	THIS^.assertorContainer.assertor.assert.strings.unicode.lengthIsExact(
		stringToCheck := stringToTest,
		expectedLength := expectedLength,
		stringLengthUnit := CNM_AssertionInterfaces.UnicodeStringLengthUnit.CHARACTERS_NFC,
		message			:= ''
	);
	
	THIS^.AssertEquals_BOOL(
		Expected 	:= assertionIsWrong,
		Actual 		:= THIS^.assertorContainer.wasAssertionWrong,
		Message 	:= messageStringBuilder.sOut
	);

	THIS^.AssertEquals_WSTRING(
		Expected 	:= stringToTestBeforeAssertion,
		Actual 		:= stringToTest,
		Message 	:= 'the assertion changed $'stringToTest$''
	);
	
CNM_AssertionInterfaces.UnicodeStringLengthUnit.VISIBLE_CHARACTERS:	
	currentStringLengthUnit := 'VISIBLE_CHARACTERS';
	
	assertionIsWrong := stringToTestVisibleCharacters <> expectedLength;
	
	message := SEL(
		assertionIsWrong,
		'stringToCheck is $'%s$' with expectedLength %u assertion must be TRUE  (%S)', 
		'stringToCheck is $'%s$' with expectedLength %u assertion must be FALSE  (%S)'
	);
	
	messageStringBuilder(
		sFormat := message,
		arg1 := THIS^.AnyToArg(stringToTestAsString),
		arg2 := THIS^.AnyToArg(expectedLength),
		arg3 := THIS^.AnyToArg(currentStringLengthUnit)
	);
	
	THIS^.assertorContainer.assertor.assert.strings.unicode.lengthIsExact(
		stringToCheck := stringToTest,
		expectedLength := expectedLength,
		stringLengthUnit := CNM_AssertionInterfaces.UnicodeStringLengthUnit.VISIBLE_CHARACTERS,
		message			:= ''
	);
	
	THIS^.AssertEquals_BOOL(
		Expected 	:= assertionIsWrong,
		Actual 		:= THIS^.assertorContainer.wasAssertionWrong,
		Message 	:= messageStringBuilder.sOut
	);

	THIS^.AssertEquals_WSTRING(
		Expected 	:= stringToTestBeforeAssertion,
		Actual 		:= stringToTest,
		Message 	:= 'the assertion changed $'stringToTest$''
	);
	
CNM_AssertionInterfaces.UnicodeStringLengthUnit.WIDTH:	
	currentStringLengthUnit := 'WIDTH';
	
	assertionIsWrong := TO_UDINT(stringToTestWidth) <> expectedLength;
	
	message := SEL(
		assertionIsWrong,
		'stringToCheck is $'%s$' with expectedLength %u assertion must be TRUE  (%S)', 
		'stringToCheck is $'%s$' with expectedLength %u assertion must be FALSE  (%S)'
	);
	
	messageStringBuilder(
		sFormat := message,
		arg1 := THIS^.AnyToArg(stringToTestAsString),
		arg2 := THIS^.AnyToArg(expectedLength),
		arg3 := THIS^.AnyToArg(currentStringLengthUnit)
	);
	
	THIS^.assertorContainer.assertor.assert.strings.unicode.lengthIsExact(
		stringToCheck := stringToTest,
		expectedLength := expectedLength,
		stringLengthUnit := CNM_AssertionInterfaces.UnicodeStringLengthUnit.WIDTH,
		message			:= ''
	);
	
	THIS^.AssertEquals_BOOL(
		Expected 	:= assertionIsWrong,
		Actual 		:= THIS^.assertorContainer.wasAssertionWrong,
		Message 	:= messageStringBuilder.sOut
	);

	THIS^.AssertEquals_WSTRING(
		Expected 	:= stringToTestBeforeAssertion,
		Actual 		:= stringToTest,
		Message 	:= 'the assertion changed $'stringToTest$''
	);

END_CASE
END_METHOD

(*
short summary
==================
This test method tests ``assert.string.unicode.lengthIsMax``
method of CNM_AssertionInterfaces library with various inputs

.. <legal notes>

legal notes
=================
| SPDX-FileCopyrightText: © 2022 ekvip automation GmbH <info@ekvip.de>
| SPDX-License-Identifier: Apache-2.0
| For details check: Apache-2.0_

.. _Apache-2.0: https://www.apache.org/licenses/LICENSE-2.0

.. </legal notes>

*)


METHOD testLengthIsMax : BOOL
VAR_INPUT
	(* for the test it's the parameter ``stringToCheck`` *)
	stringToTest 			:WSTRING(Tc2_System.MAX_STRING_LENGTH);
	(* for the test it's the parameter ``maxLength`` *)
	expectedLength 			:UDINT;
	(* UnicodeStringLengthUnit the input is tested for *)
	stringLengthUnit		:CNM_AssertionInterfaces.UnicodeStringLengthUnit;
	(* contains ``stringToTest`` in only ascii charachters for test output *)
	stringToTestPrintable	:Tc2_System.T_MaxString := '';
END_VAR
VAR 
	(* just the expectation if the assertion to test must be worng or true *)
	assertionIsWrong					:BOOL;
	(* contains the format string for the test message *)
	message								:Tc2_System.T_MaxString;
	(* used for placeholder string if stringToTest can't be printed *)
	stringToTestAsString 				:Tc2_System.T_MaxString;
	(* holds string with current ´´stringLengthUnit´´ for the test message*)
	currentStringLengthUnit 			:Tc2_System.T_MaxString;
	(* TwinCAT printf with the test message *)
	messageStringBuilder				:Tc2_Utilities.FB_FormatString;
	(* length of current string to check in bytes *)
	stringToTestByteCount				:UDINT;
	(* count of words in current string *)
	stringToTestWordCount				:UDINT;
	(* length of current string to check in characters *)
	stringToTestCodePointCount			:UDINT;
	(* length of ´´stringToCheck´´ *)
	normalizedLength 					:UDINT;
	(* holds the normalized ´´stringToCheck´´ *)
	normalizedStringToTest 				:WSTRING(Tc2_System.MAX_STRING_LENGTH);
	(* width of ´´stringToCheck´´ *)
	stringToTestWidth 					:DINT;
	(* visible characters of ´´stringToCheck´´ *)
	stringToTestVisibleCharacters 		:UDINT := 0;
	(*string in UTF32*)
	utf32String							:ARRAY [0..Tc2_System.Global_Variables.MAX_STRING_LENGTH]  OF CNM_UnicodeUtilities.UnicodeCodePoint;
	(* utf32 code point count *)
	utf32CodePointCount 				:UDINT;
	(* bytes in utf8 string *)
	utf8ByteCount 						:UDINT;
	(* hold stringToCheck before assertion *)
	stringToTestBeforeAssertion			:WSTRING(Tc2_System.MAX_STRING_LENGTH);
END_VAR
THIS^.assertorContainer.resetAssertor();

stringToTestBeforeAssertion := stringToTest;

CNM_UnicodeUtilities.GetUtf16StringLength(ADR(stringToTest), wordCount => stringToTestWordCount, characterCount => stringToTestCodePointCount,);
CNM_UnicodeUtilities.GetUtf16StringWidth(ADR(stringToTest), visibleCharacters => stringToTestVisibleCharacters, width => stringToTestWidth);
stringToTestByteCount := stringToTestWordCount * 2;

CNM_UnicodeUtilities.GetCodepointsFromUtf16String(
	utf16StringAddress := ADR(stringToTest),
	utf16StringWordCount := stringToTestWordCount,
	codepointBuffer :=ADR(utf32String),
	bufferSize := SIZEOF(utf32String),
	codePointCount => utf32CodePointCount
);

CNM_UnicodeUtilities.GetUtf8StringFromCodepoints(
	addressOfCodePoints := ADR(utf32String),
	codePointCount := utf32CodePointCount,
	utf8StringBuffer := ADR(stringToTestAsString),
	bufferSize := MAX_STRING_LENGTH + 1,
	utf8StringByteCount => utf8ByteCount
);

IF ( Tc2_Standard.LEN(stringToTestPrintable) <> 0 ) THEN
	stringToTestAsString := stringToTestPrintable;
END_IF


CASE stringLengthUnit OF
	
CNM_AssertionInterfaces.UnicodeStringLengthUnit.BYTES:
	currentStringLengthUnit := 'BYTES';
	
	assertionIsWrong := stringToTestByteCount > expectedLength;
	
	message := SEL(
		assertionIsWrong,
		'stringToCheck is $'%s$' with expectedLength %u assertion must be TRUE  (%S)', 
		'stringToCheck is $'%s$' with expectedLength %u assertion must be FALSE  (%S)'
	);
	
	messageStringBuilder(
		sFormat := message,
		arg1 := THIS^.AnyToArg(stringToTestAsString),
		arg2 := THIS^.AnyToArg(expectedLength),
		arg3 := THIS^.AnyToArg(currentStringLengthUnit)
	);
	
	THIS^.assertorContainer.assertor.assert.strings.unicode.lengthIsMax(
		stringToCheck := stringToTest,
		maxLength := expectedLength,
		stringLengthUnit := CNM_AssertionInterfaces.UnicodeStringLengthUnit.BYTES,
		message			:= ''
	);
	
	THIS^.AssertEquals_BOOL(
		Expected 	:= assertionIsWrong,
		Actual 		:= THIS^.assertorContainer.wasAssertionWrong,
		Message 	:= messageStringBuilder.sOut
	);

	THIS^.AssertEquals_WSTRING(
		Expected 	:= stringToTestBeforeAssertion,
		Actual 		:= stringToTest,
		Message 	:= 'the assertion changed $'stringToTest$''
	);
	
CNM_AssertionInterfaces.UnicodeStringLengthUnit.CHARACTERS:	
	currentStringLengthUnit := 'CHARACTERS';
	
	assertionIsWrong := stringToTestCodePointCount > expectedLength;
	
	message := SEL(
		assertionIsWrong,
		'stringToCheck is $'%s$' with expectedLength %u assertion must be TRUE  (%S)', 
		'stringToCheck is $'%s$' with expectedLength %u assertion must be FALSE  (%S)'
	);
	
	messageStringBuilder(
		sFormat := message,
		arg1 := THIS^.AnyToArg(stringToTestAsString),
		arg2 := THIS^.AnyToArg(expectedLength),
		arg3 := THIS^.AnyToArg(currentStringLengthUnit)
	);
	
	THIS^.assertorContainer.assertor.assert.strings.unicode.lengthIsMax(
		stringToCheck := stringToTest,
		maxLength := expectedLength,
		stringLengthUnit := CNM_AssertionInterfaces.UnicodeStringLengthUnit.CHARACTERS,
		message			:= ''
	);
	
	THIS^.AssertEquals_BOOL(
		Expected 	:= assertionIsWrong,
		Actual 		:= THIS^.assertorContainer.wasAssertionWrong,
		Message 	:= messageStringBuilder.sOut
	);

	THIS^.AssertEquals_WSTRING(
		Expected 	:= stringToTestBeforeAssertion,
		Actual 		:= stringToTest,
		Message 	:= 'the assertion changed $'stringToTest$''
	);
	
CNM_AssertionInterfaces.UnicodeStringLengthUnit.CHARACTERS_NFD:	
	currentStringLengthUnit := 'NFD';
	
	CNM_UnicodeUtilities.NormalizeUtf16String(
		utf16StringBuffer := ADR(stringToTest),
		normalForm := CNM_UnicodeUtilities.NormalizationForm.NFD,
		normalizedStringBuffer := ADR(normalizedStringToTest),
		bufferSize := Tc2_System.MAX_STRING_LENGTH * 2 + 2,
		normalizedStringLength => normalizedLength
	);
	CNM_UnicodeUtilities.GetUtf16StringLength(
		utf16StringAddress := ADR(normalizedStringToTest),
		characterCount => stringToTestCodePointCount
	);
		
	assertionIsWrong := stringToTestCodePointCount > expectedLength;
	
	message := SEL(
		assertionIsWrong,
		'stringToCheck is $'%s$' with expectedLength %u assertion must be TRUE  (%S)', 
		'stringToCheck is $'%s$' with expectedLength %u assertion must be FALSE  (%S)'
	);
	
	messageStringBuilder(
		sFormat := message,
		arg1 := THIS^.AnyToArg(stringToTestAsString),
		arg2 := THIS^.AnyToArg(expectedLength),
		arg3 := THIS^.AnyToArg(currentStringLengthUnit)
	);
	
	THIS^.assertorContainer.assertor.assert.strings.unicode.lengthIsMax(
		stringToCheck := stringToTest,
		maxLength := expectedLength,
		stringLengthUnit := CNM_AssertionInterfaces.UnicodeStringLengthUnit.CHARACTERS_NFD,
		message			:= ''
	);
	
	THIS^.AssertEquals_BOOL(
		Expected 	:= assertionIsWrong,
		Actual 		:= THIS^.assertorContainer.wasAssertionWrong,
		Message 	:= messageStringBuilder.sOut
	);

	THIS^.AssertEquals_WSTRING(
		Expected 	:= stringToTestBeforeAssertion,
		Actual 		:= stringToTest,
		Message 	:= 'the assertion changed $'stringToTest$''
	);
	
CNM_AssertionInterfaces.UnicodeStringLengthUnit.CHARACTERS_NFC:	
	currentStringLengthUnit := 'NFC';
	
	CNM_UnicodeUtilities.NormalizeUtf16String(
		utf16StringBuffer := ADR(stringToTest),
		normalForm := CNM_UnicodeUtilities.NormalizationForm.NFC,
		normalizedStringBuffer := ADR(normalizedStringToTest),
		bufferSize := Tc2_System.MAX_STRING_LENGTH * 2 + 2,
		normalizedStringLength => normalizedLength
	);
	CNM_UnicodeUtilities.GetUtf16StringLength(
		utf16StringAddress := ADR(normalizedStringToTest),
		characterCount => stringToTestCodePointCount
	);
		
	assertionIsWrong := stringToTestCodePointCount > expectedLength;
	
	message := SEL(
		assertionIsWrong,
		'stringToCheck is $'%s$' with expectedLength %u assertion must be TRUE  (%S)', 
		'stringToCheck is $'%s$' with expectedLength %u assertion must be FALSE  (%S)'
	);
	
	messageStringBuilder(
		sFormat := message,
		arg1 := THIS^.AnyToArg(stringToTestAsString),
		arg2 := THIS^.AnyToArg(expectedLength),
		arg3 := THIS^.AnyToArg(currentStringLengthUnit)
	);
	
	THIS^.assertorContainer.assertor.assert.strings.unicode.lengthIsMax(
		stringToCheck := stringToTest,
		maxLength := expectedLength,
		stringLengthUnit := CNM_AssertionInterfaces.UnicodeStringLengthUnit.CHARACTERS_NFC,
		message			:= ''
	);
	
	THIS^.AssertEquals_BOOL(
		Expected 	:= assertionIsWrong,
		Actual 		:= THIS^.assertorContainer.wasAssertionWrong,
		Message 	:= messageStringBuilder.sOut
	);

	THIS^.AssertEquals_WSTRING(
		Expected 	:= stringToTestBeforeAssertion,
		Actual 		:= stringToTest,
		Message 	:= 'the assertion changed $'stringToTest$''
	);
	
CNM_AssertionInterfaces.UnicodeStringLengthUnit.VISIBLE_CHARACTERS:	
	currentStringLengthUnit := 'VISIBLE_CHARACTERS';
	
	assertionIsWrong := stringToTestVisibleCharacters > expectedLength;
	
	message := SEL(
		assertionIsWrong,
		'stringToCheck is $'%s$' with expectedLength %u assertion must be TRUE  (%S)', 
		'stringToCheck is $'%s$' with expectedLength %u assertion must be FALSE  (%S)'
	);
	
	messageStringBuilder(
		sFormat := message,
		arg1 := THIS^.AnyToArg(stringToTestAsString),
		arg2 := THIS^.AnyToArg(expectedLength),
		arg3 := THIS^.AnyToArg(currentStringLengthUnit)
	);
	
	THIS^.assertorContainer.assertor.assert.strings.unicode.lengthIsMax(
		stringToCheck := stringToTest,
		maxLength := expectedLength,
		stringLengthUnit := CNM_AssertionInterfaces.UnicodeStringLengthUnit.VISIBLE_CHARACTERS,
		message			:= ''
	);
	
	THIS^.AssertEquals_BOOL(
		Expected 	:= assertionIsWrong,
		Actual 		:= THIS^.assertorContainer.wasAssertionWrong,
		Message 	:= messageStringBuilder.sOut
	);

	THIS^.AssertEquals_WSTRING(
		Expected 	:= stringToTestBeforeAssertion,
		Actual 		:= stringToTest,
		Message 	:= 'the assertion changed $'stringToTest$''
	);
	
CNM_AssertionInterfaces.UnicodeStringLengthUnit.WIDTH:	
	currentStringLengthUnit := 'WIDTH';
	
	assertionIsWrong := TO_UDINT(stringToTestWidth) > expectedLength;
	
	message := SEL(
		assertionIsWrong,
		'stringToCheck is $'%s$' with expectedLength %u assertion must be TRUE  (%S)', 
		'stringToCheck is $'%s$' with expectedLength %u assertion must be FALSE  (%S)'
	);
	
	messageStringBuilder(
		sFormat := message,
		arg1 := THIS^.AnyToArg(stringToTestAsString),
		arg2 := THIS^.AnyToArg(expectedLength),
		arg3 := THIS^.AnyToArg(currentStringLengthUnit)
	);
	
	THIS^.assertorContainer.assertor.assert.strings.unicode.lengthIsMax(
		stringToCheck := stringToTest,
		maxLength := expectedLength,
		stringLengthUnit := CNM_AssertionInterfaces.UnicodeStringLengthUnit.WIDTH,
		message			:= ''
	);
	
	THIS^.AssertEquals_BOOL(
		Expected 	:= assertionIsWrong,
		Actual 		:= THIS^.assertorContainer.wasAssertionWrong,
		Message 	:= messageStringBuilder.sOut
	);

	THIS^.AssertEquals_WSTRING(
		Expected 	:= stringToTestBeforeAssertion,
		Actual 		:= stringToTest,
		Message 	:= 'the assertion changed $'stringToTest$''
	);

END_CASE
END_METHOD

(*
short summary
==================
This test method tests ``assert.string.unicode.lengthIsMin``
method of CNM_AssertionInterfaces library with various inputs

.. <legal notes>

legal notes
=================
| SPDX-FileCopyrightText: © 2022 ekvip automation GmbH <info@ekvip.de>
| SPDX-License-Identifier: Apache-2.0
| For details check: Apache-2.0_

.. _Apache-2.0: https://www.apache.org/licenses/LICENSE-2.0

.. </legal notes>

*)


METHOD testLengthIsMin : BOOL
VAR_INPUT
	(* for the test it's the parameter ``stringToCheck`` *)
	stringToTest 			:WSTRING(Tc2_System.MAX_STRING_LENGTH);
	(* for the test it's the parameter ``minLength`` *)
	expectedLength 			:UDINT;
	(* UnicodeStringLengthUnit the input is tested for *)
	stringLengthUnit		:CNM_AssertionInterfaces.UnicodeStringLengthUnit;
	(* contains ``stringToTest`` in only ascii charachters for test output *)
	stringToTestPrintable	:Tc2_System.T_MaxString := '';
END_VAR
VAR 
	(* just the expectation if the assertion to test must be worng or true *)
	assertionIsWrong				:BOOL;
	(* contains the format string for the test message *)
	message							:Tc2_System.T_MaxString;
	(* used for placeholder string if stringToTest can't be printed *)
	stringToTestAsString 			:Tc2_System.T_MaxString;
	(* holds string with current ´´stringLengthUnit´´ for the test message*)
	currentStringLengthUnit 		:Tc2_System.T_MaxString;
	(* TwinCAT printf with the test message *)
	messageStringBuilder			:Tc2_Utilities.FB_FormatString;
	(* length of current string to check in bytes *)
	stringToTestByteCount			:UDINT;
	(* count of words in current string *)
	stringToTestWordCount			:UDINT;
	(* length of current string to check in characters *)
	stringToTestCodePointCount		:UDINT;
	(* length of ´´stringToCheck´´ *)
	normalizedLength 				:UDINT;
	(* holds the normalized ´´stringToCheck´´ *)
	normalizedStringToTest 			:WSTRING(Tc2_System.MAX_STRING_LENGTH);
	(* width of ´´stringToCheck´´ *)
	stringToTestWidth 				:DINT;
	(* visible characters of ´´stringToCheck´´ *)
	stringToTestVisibleCharacters 	:UDINT := 0;
	(*string in UTF32*)
	utf32String						:ARRAY [0..Tc2_System.Global_Variables.MAX_STRING_LENGTH]  OF CNM_UnicodeUtilities.UnicodeCodePoint;
	(* utf32 code point count *)
	utf32CodePointCount 			:UDINT;
	(* bytes in utf8 string *)
	utf8ByteCount 					:UDINT;
	(* hold stringToCheck before assertion *)
	stringToTestBeforeAssertion		:WSTRING(Tc2_System.MAX_STRING_LENGTH);
END_VAR
THIS^.assertorContainer.resetAssertor();

stringToTestBeforeAssertion := stringToTest;

CNM_UnicodeUtilities.GetUtf16StringLength(ADR(stringToTest), wordCount => stringToTestWordCount, characterCount => stringToTestCodePointCount,);
CNM_UnicodeUtilities.GetUtf16StringWidth(ADR(stringToTest), visibleCharacters => stringToTestVisibleCharacters, width => stringToTestWidth);
stringToTestByteCount := stringToTestWordCount * 2;

CNM_UnicodeUtilities.GetCodepointsFromUtf16String(
	utf16StringAddress := ADR(stringToTest),
	utf16StringWordCount := stringToTestWordCount,
	codepointBuffer :=ADR(utf32String),
	bufferSize := SIZEOF(utf32String),
	codePointCount => utf32CodePointCount
);

CNM_UnicodeUtilities.GetUtf8StringFromCodepoints(
	addressOfCodePoints := ADR(utf32String),
	codePointCount := utf32CodePointCount,
	utf8StringBuffer := ADR(stringToTestAsString),
	bufferSize := MAX_STRING_LENGTH + 1,
	utf8StringByteCount => utf8ByteCount
);

IF ( Tc2_Standard.LEN(stringToTestPrintable) <> 0 ) THEN
	stringToTestAsString := stringToTestPrintable;
END_IF


CASE stringLengthUnit OF
	
CNM_AssertionInterfaces.UnicodeStringLengthUnit.BYTES:	
	currentStringLengthUnit := 'BYTES';
	
	assertionIsWrong := stringToTestByteCount < expectedLength;
	
	message := SEL(
		assertionIsWrong,
		'stringToCheck is $'%s$' with expectedLength %u assertion must be TRUE  (%S)', 
		'stringToCheck is $'%s$' with expectedLength %u assertion must be FALSE  (%S)'
	);
	
	messageStringBuilder(
		sFormat := message,
		arg1 := THIS^.AnyToArg(stringToTestAsString),
		arg2 := THIS^.AnyToArg(expectedLength),
		arg3 := THIS^.AnyToArg(currentStringLengthUnit)
	);
	
	THIS^.assertorContainer.assertor.assert.strings.unicode.lengthIsMin(
		stringToCheck := stringToTest,
		minLength := expectedLength,
		stringLengthUnit := CNM_AssertionInterfaces.UnicodeStringLengthUnit.BYTES,
		message			:= ''
	);
	
	THIS^.AssertEquals_BOOL(
		Expected 	:= assertionIsWrong,
		Actual 		:= THIS^.assertorContainer.wasAssertionWrong,
		Message 	:= messageStringBuilder.sOut
	);

	THIS^.AssertEquals_WSTRING(
		Expected 	:= stringToTestBeforeAssertion,
		Actual 		:= stringToTest,
		Message 	:= 'the assertion changed $'stringToTest$''
	);
	
CNM_AssertionInterfaces.UnicodeStringLengthUnit.CHARACTERS:	
	currentStringLengthUnit := 'CHARACTERS';
	
	assertionIsWrong := stringToTestCodePointCount < expectedLength;
	
	message := SEL(
		assertionIsWrong,
		'stringToCheck is $'%s$' with expectedLength %u assertion must be TRUE  (%S)', 
		'stringToCheck is $'%s$' with expectedLength %u assertion must be FALSE  (%S)'
	);
	
	messageStringBuilder(
		sFormat := message,
		arg1 := THIS^.AnyToArg(stringToTestAsString),
		arg2 := THIS^.AnyToArg(expectedLength),
		arg3 := THIS^.AnyToArg(currentStringLengthUnit)
	);
	
	THIS^.assertorContainer.assertor.assert.strings.unicode.lengthIsMin(
		stringToCheck := stringToTest,
		minLength := expectedLength,
		stringLengthUnit := CNM_AssertionInterfaces.UnicodeStringLengthUnit.CHARACTERS,
		message			:= ''
	);
	
	THIS^.AssertEquals_BOOL(
		Expected 	:= assertionIsWrong,
		Actual 		:= THIS^.assertorContainer.wasAssertionWrong,
		Message 	:= messageStringBuilder.sOut
	);

	THIS^.AssertEquals_WSTRING(
		Expected 	:= stringToTestBeforeAssertion,
		Actual 		:= stringToTest,
		Message 	:= 'the assertion changed $'stringToTest$''
	);
	
CNM_AssertionInterfaces.UnicodeStringLengthUnit.CHARACTERS_NFD:	
	currentStringLengthUnit := 'NFD';
	
	CNM_UnicodeUtilities.NormalizeUtf16String(
		utf16StringBuffer := ADR(stringToTest),
		normalForm := CNM_UnicodeUtilities.NormalizationForm.NFD,
		normalizedStringBuffer := ADR(normalizedStringToTest),
		bufferSize := Tc2_System.MAX_STRING_LENGTH * 2 + 2,
		normalizedStringLength => normalizedLength
	);
	CNM_UnicodeUtilities.GetUtf16StringLength(
		utf16StringAddress := ADR(normalizedStringToTest),
		characterCount => stringToTestCodePointCount
	);
		
	assertionIsWrong := stringToTestCodePointCount < expectedLength;
	
	message := SEL(
		assertionIsWrong,
		'stringToCheck is $'%s$' with expectedLength %u assertion must be TRUE  (%S)', 
		'stringToCheck is $'%s$' with expectedLength %u assertion must be FALSE  (%S)'
	);
	
	messageStringBuilder(
		sFormat := message,
		arg1 := THIS^.AnyToArg(stringToTestAsString),
		arg2 := THIS^.AnyToArg(expectedLength),
		arg3 := THIS^.AnyToArg(currentStringLengthUnit)
	);
	
	THIS^.assertorContainer.assertor.assert.strings.unicode.lengthIsMin(
		stringToCheck := stringToTest,
		minLength := expectedLength,
		stringLengthUnit := CNM_AssertionInterfaces.UnicodeStringLengthUnit.CHARACTERS_NFD,
		message			:= ''
	);
	
	THIS^.AssertEquals_BOOL(
		Expected 	:= assertionIsWrong,
		Actual 		:= THIS^.assertorContainer.wasAssertionWrong,
		Message 	:= messageStringBuilder.sOut
	);

	THIS^.AssertEquals_WSTRING(
		Expected 	:= stringToTestBeforeAssertion,
		Actual 		:= stringToTest,
		Message 	:= 'the assertion changed $'stringToTest$''
	);
	
CNM_AssertionInterfaces.UnicodeStringLengthUnit.CHARACTERS_NFC:	
	currentStringLengthUnit := 'NFC';
	
	CNM_UnicodeUtilities.NormalizeUtf16String(
		utf16StringBuffer := ADR(stringToTest),
		normalForm := CNM_UnicodeUtilities.NormalizationForm.NFC,
		normalizedStringBuffer := ADR(normalizedStringToTest),
		bufferSize := Tc2_System.MAX_STRING_LENGTH * 2 + 2,
		normalizedStringLength => normalizedLength
	);
	CNM_UnicodeUtilities.GetUtf16StringLength(
		utf16StringAddress := ADR(normalizedStringToTest),
		characterCount => stringToTestCodePointCount
	);
		
	assertionIsWrong := stringToTestCodePointCount < expectedLength;
	
	message := SEL(
		assertionIsWrong,
		'stringToCheck is $'%s$' with expectedLength %u assertion must be TRUE  (%S)', 
		'stringToCheck is $'%s$' with expectedLength %u assertion must be FALSE  (%S)'
	);
	
	messageStringBuilder(
		sFormat := message,
		arg1 := THIS^.AnyToArg(stringToTestAsString),
		arg2 := THIS^.AnyToArg(expectedLength),
		arg3 := THIS^.AnyToArg(currentStringLengthUnit)
	);
	
	THIS^.assertorContainer.assertor.assert.strings.unicode.lengthIsMin(
		stringToCheck := stringToTest,
		minLength := expectedLength,
		stringLengthUnit := CNM_AssertionInterfaces.UnicodeStringLengthUnit.CHARACTERS_NFC,
		message			:= ''
	);
	
	THIS^.AssertEquals_BOOL(
		Expected 	:= assertionIsWrong,
		Actual 		:= THIS^.assertorContainer.wasAssertionWrong,
		Message 	:= messageStringBuilder.sOut
	);
	
	THIS^.AssertEquals_WSTRING(
		Expected 	:= stringToTestBeforeAssertion,
		Actual 		:= stringToTest,
		Message 	:= 'the assertion changed $'stringToTest$''
	);

CNM_AssertionInterfaces.UnicodeStringLengthUnit.VISIBLE_CHARACTERS:	
	currentStringLengthUnit := 'VISIBLE_CHARACTERS';
	
	assertionIsWrong := stringToTestVisibleCharacters < expectedLength;
	
	message := SEL(
		assertionIsWrong,
		'stringToCheck is $'%s$' with expectedLength %u assertion must be TRUE  (%S)', 
		'stringToCheck is $'%s$' with expectedLength %u assertion must be FALSE  (%S)'
	);
	
	messageStringBuilder(
		sFormat := message,
		arg1 := THIS^.AnyToArg(stringToTestAsString),
		arg2 := THIS^.AnyToArg(expectedLength),
		arg3 := THIS^.AnyToArg(currentStringLengthUnit)
	);
	
	THIS^.assertorContainer.assertor.assert.strings.unicode.lengthIsMin(
		stringToCheck := stringToTest,
		minLength := expectedLength,
		stringLengthUnit := CNM_AssertionInterfaces.UnicodeStringLengthUnit.VISIBLE_CHARACTERS,
		message			:= ''
	);
	
	THIS^.AssertEquals_BOOL(
		Expected 	:= assertionIsWrong,
		Actual 		:= THIS^.assertorContainer.wasAssertionWrong,
		Message 	:= messageStringBuilder.sOut
	);
	
	THIS^.AssertEquals_WSTRING(
		Expected 	:= stringToTestBeforeAssertion,
		Actual 		:= stringToTest,
		Message 	:= 'the assertion changed $'stringToTest$''
	);

CNM_AssertionInterfaces.UnicodeStringLengthUnit.WIDTH:	
	currentStringLengthUnit := 'WIDTH';
	
	assertionIsWrong := TO_UDINT(stringToTestWidth) < expectedLength;
	
	message := SEL(
		assertionIsWrong,
		'stringToCheck is $'%s$' with expectedLength %u assertion must be TRUE  (%S)', 
		'stringToCheck is $'%s$' with expectedLength %u assertion must be FALSE  (%S)'
	);
	
	messageStringBuilder(
		sFormat := message,
		arg1 := THIS^.AnyToArg(stringToTestAsString),
		arg2 := THIS^.AnyToArg(expectedLength),
		arg3 := THIS^.AnyToArg(currentStringLengthUnit)
	);
	
	THIS^.assertorContainer.assertor.assert.strings.unicode.lengthIsMin(
		stringToCheck := stringToTest,
		minLength := expectedLength,
		stringLengthUnit := CNM_AssertionInterfaces.UnicodeStringLengthUnit.WIDTH,
		message			:= ''
	);
	
	THIS^.AssertEquals_BOOL(
		Expected 	:= assertionIsWrong,
		Actual 		:= THIS^.assertorContainer.wasAssertionWrong,
		Message 	:= messageStringBuilder.sOut
	);

	THIS^.AssertEquals_WSTRING(
		Expected 	:= stringToTestBeforeAssertion,
		Actual 		:= stringToTest,
		Message 	:= 'the assertion changed $'stringToTest$''
	);

END_CASE
END_METHOD

(*
short summary
==================
This test method tests ``assert.string.unicode.startsWith``
method of CNM_AssertionInterfaces library with various inputs

.. <legal notes>

legal notes
=================
| SPDX-FileCopyrightText: © 2022 ekvip automation GmbH <info@ekvip.de>
| SPDX-License-Identifier: Apache-2.0
| For details check: Apache-2.0_

.. _Apache-2.0: https://www.apache.org/licenses/LICENSE-2.0

.. </legal notes>

*)


METHOD testStartsWith : BOOL
VAR_INPUT
	(* for the test it's the parameter ``stringToCheck`` *)
	stringToTest  	:WSTRING(Tc2_System.MAX_STRING_LENGTH);
	(* for the test it's the parameter ``searchString`` *)
	expectedString	:WSTRING(Tc2_System.MAX_STRING_LENGTH);
END_VAR
VAR 
	(* just the expectation if the assertion to test must be worng or true *)
	assertionIsWrong				:BOOL;
	(* contains the format string for the test message *)
	message							:Tc2_System.T_MaxString;
	(* used for placeholder string if stringToTest can't be printed *)
	stringToTestAsString 			:Tc2_System.T_MaxString;
	(* used for placeholder string if expectedString can't be printed *)
	expectedStringAsString 			:Tc2_System.T_MaxString;
	(* contains stringToTest in normalized form *)
	normalizedStringToTest			:WSTRING(Tc2_System.MAX_STRING_LENGTH);
	(* contains expectedString in normalized form *)
	normalizedExpectedString		:WSTRING(Tc2_System.MAX_STRING_LENGTH);
	(* holds characterCount of ``expectedString`` *)
	expectedCharacterCount			:UDINT;
	(* TwinCAT printf with the test message *)
	messageStringBuilder			:Tc2_Utilities.FB_FormatString;
	(* hold stringToCheck before assertion *)
	stringToTestBeforeAssertion		:WSTRING(Tc2_System.MAX_STRING_LENGTH);
	(* hold stringToCheck before assertion *)
	expectedStringBeforeAssertion	:WSTRING(Tc2_System.MAX_STRING_LENGTH);
END_VAR
THIS^.assertorContainer.resetAssertor();

stringToTestBeforeAssertion := stringToTest;
expectedStringBeforeAssertion := expectedString;

CNM_UnicodeUtilities.GetUtf16StringLength(
	utf16StringAddress := ADR(expectedString),
	characterCount => expectedCharacterCount
);
assertionIsWrong := ((
		CNM_UnicodeUtilities.FindInUtf16String(
			ADR(stringToTest),
			ADR(expectedString),
		) <> 1
	) AND (
		expectedCharacterCount <> 0
	)
);

message := SEL(
	assertionIsWrong,
	'stringToCheck is $'%s$' start is $'%s$' assertion must be TRUE', 
	'stringToCheck is $'%s$' start is $'%s$' assertion must be FALSE'
);

Tc2_Utilities.WSTRING_TO_STRING2(ADR(stringToTestAsString), ADR(stringToTest), SIZEOF(stringToTestAsString));
Tc2_Utilities.WSTRING_TO_STRING2(ADR(expectedStringAsString), ADR(expectedString), SIZEOF(expectedStringAsString));

IF (
		Tc2_Standard.WLEN(stringToTest) = TO_UINT(Tc2_System.MAX_STRING_LENGTH)
) THEN
	stringToTestAsString := 'String with Tc2_System.MAX_STRING_LENGTH characters';
END_IF
IF (
		Tc2_Standard.WLEN(expectedString) = TO_UINT(Tc2_System.MAX_STRING_LENGTH)
) THEN
	expectedStringAsString := 'String with Tc2_System.MAX_STRING_LENGTH characters';
END_IF

messageStringBuilder(
	sFormat := message,
	arg1 := THIS^.AnyToArg(stringToTestAsString),
	arg2 := THIS^.AnyToArg(expectedStringAsString)
);


THIS^.assertorContainer.assertor.assert.strings.unicode.startsWith(
	stringToCheck := stringToTest,
	start := expectedString,
	ignoreCases := FALSE,
	trim := FALSE,
	normalizeStrings := FALSE,
	message			:= ''
);

THIS^.AssertEquals_BOOL(
	Expected 	:= assertionIsWrong,
	Actual 		:= THIS^.assertorContainer.wasAssertionWrong,
	Message 	:= messageStringBuilder.sOut
);

THIS^.AssertEquals_WSTRING(
	Expected 	:= stringToTestBeforeAssertion,
	Actual 		:= stringToTest,
	Message 	:= 'the assertion changed $'stringToTest$''
);

THIS^.AssertEquals_WSTRING(
	Expected 	:= expectedStringBeforeAssertion,
	Actual 		:= expectedString,
	Message 	:= 'the assertion changed $'expectedString$''
);

THIS^.assertorContainer.resetAssertor();

CNM_UnicodeUtilities.NormalizeUtf16String(
	utf16StringBuffer := ADR(stringToTest),
	bufferSize := Tc2_System.MAX_STRING_LENGTH * 2 + 2,
	normalizedStringBuffer := ADR(normalizedStringToTest),
	normalForm := CNM_UnicodeUtilities.NormalizationForm.NFD
);
CNM_UnicodeUtilities.NormalizeUtf16String(
	utf16StringBuffer := ADR(expectedString),
	bufferSize := Tc2_System.MAX_STRING_LENGTH * 2 + 2,
	normalizedStringBuffer := ADR(normalizedExpectedString),
	normalForm := CNM_UnicodeUtilities.NormalizationForm.NFD
);

CNM_UnicodeUtilities.GetUtf16StringLength(
	utf16StringAddress := ADR(normalizedExpectedString),
	characterCount => expectedCharacterCount
);
// no trim for ``start`` expected
assertionIsWrong := ((
		CNM_UnicodeUtilities.FindInUtf16String(
			ADR(normalizedStringToTest),
			ADR(normalizedExpectedString),
		) <> 1
	) AND (
		expectedCharacterCount <> 0
	)
);

THIS^.assertorContainer.assertor.assert.strings.unicode.startsWith(
	stringToCheck := stringToTest,
	start := expectedString,
	ignoreCases := FALSE,
	trim		:= FALSE,
	normalizeStrings := TRUE,
	message			:= ''
);

THIS^.AssertEquals_BOOL(
	Expected 	:= assertionIsWrong,
	Actual 		:= THIS^.assertorContainer.wasAssertionWrong,
	Message 	:= messageStringBuilder.sOut
);

THIS^.AssertEquals_WSTRING(
	Expected 	:= stringToTestBeforeAssertion,
	Actual 		:= stringToTest,
	Message 	:= 'the assertion changed $'stringToTest$''
);

THIS^.AssertEquals_WSTRING(
	Expected 	:= expectedStringBeforeAssertion,
	Actual 		:= expectedString,
	Message 	:= 'the assertion changed $'expectedString$''
);
END_METHOD

(*
short summary
==================
This test method tests ``assert.string.unicode.startsWith``
method of CNM_AssertionInterfaces library with various inputs

.. <legal notes>

legal notes
=================
| SPDX-FileCopyrightText: © 2022 ekvip automation GmbH <info@ekvip.de>
| SPDX-License-Identifier: Apache-2.0
| For details check: Apache-2.0_

.. _Apache-2.0: https://www.apache.org/licenses/LICENSE-2.0

.. </legal notes>

*)


METHOD testStartsWithIgnoreCase : BOOL
VAR_INPUT
	(* for the test it's the parameter ``stringToCheck`` *)
	stringToTest  	:WSTRING(Tc2_System.MAX_STRING_LENGTH);
	(* for the test it's the parameter ``searchString`` *)
	expectedString	:WSTRING(Tc2_System.MAX_STRING_LENGTH);
END_VAR
VAR 
	(* just the expectation if the assertion to test must be worng or true *)
	assertionIsWrong				:BOOL;
	(* contains the format string for the test message *)
	message							:Tc2_System.T_MaxString;
	(* contains ´´stringToTest´´ in upper case *)
	upperStringToTest				:WSTRING(Tc2_System.MAX_STRING_LENGTH);
	(* contains ´´expectedString´´ in upper case *)
	upperExpectedString				:WSTRING(Tc2_System.MAX_STRING_LENGTH);
	(* used for placeholder string if stringToTest can't be printed *)
	stringToTestAsString 			:Tc2_System.T_MaxString;
	(* used for placeholder string if expectedString can't be printed *)
	expectedStringAsString			:Tc2_System.T_MaxString;
	(* contains stringToTest in normalized form *)
	normalizedStringToTest			:WSTRING(Tc2_System.MAX_STRING_LENGTH);
	(* contains expectedString in normalized form *)
	normalizedExpectedString		:WSTRING(Tc2_System.MAX_STRING_LENGTH);
	(* contains stringToTest in normalized form in upper case*)
	normalizedUpperStringToTest		:WSTRING(Tc2_System.MAX_STRING_LENGTH);
	(* contains expectedString in normalized form in upper case*)
	normalizedUpperExpectedString	:WSTRING(Tc2_System.MAX_STRING_LENGTH);
	(* holds characterCount of ``expectedString`` *)
	expectedCharacterCount			:UDINT;
	(* TwinCAT printf with the test message *)
	messageStringBuilder			:Tc2_Utilities.FB_FormatString;
	(* hold stringToCheck before assertion *)
	stringToTestBeforeAssertion		:WSTRING(Tc2_System.MAX_STRING_LENGTH);
	(* hold stringToCheck before assertion *)
	expectedStringBeforeAssertion	:WSTRING(Tc2_System.MAX_STRING_LENGTH);
END_VAR
THIS^.assertorContainer.resetAssertor();

stringToTestBeforeAssertion := stringToTest;
expectedStringBeforeAssertion := expectedString;

upperStringToTest := stringToTest;
upperExpectedString := expectedString;

// both Strings to upper case
CNM_UnicodeUtilities.GetUpperCaseUtf16(ADR(upperStringToTest));
CNM_UnicodeUtilities.GetUpperCaseUtf16(ADR(upperExpectedString));

CNM_UnicodeUtilities.GetUtf16StringLength(
	utf16StringAddress := ADR(upperExpectedString),
	characterCount => expectedCharacterCount
);	
assertionIsWrong := ((
		CNM_UnicodeUtilities.FindInUtf16String(
			ADR(upperStringToTest),
			ADR(upperExpectedString)
		) <> 1 
	) AND (
		expectedCharacterCount <> 0
	)
);

message := SEL(
	assertionIsWrong,
	'stringToCheck is $'%s$' start is $'%s$' assertion must be TRUE', 
	'stringToCheck is $'%s$' start is $'%s$' assertion must be FALSE'
);

Tc2_Utilities.WSTRING_TO_STRING2(ADR(stringToTestAsString), ADR(stringToTest), SIZEOF(stringToTestAsString));
Tc2_Utilities.WSTRING_TO_STRING2(ADR(expectedStringAsString), ADR(expectedString), SIZEOF(expectedStringAsString));

IF (
		Tc2_Standard.WLEN(stringToTest) = TO_UINT(Tc2_System.MAX_STRING_LENGTH)
) THEN
	stringToTestAsString := 'String with Tc2_System.MAX_STRING_LENGTH characters';
END_IF
IF (
		Tc2_Standard.WLEN(expectedString) = TO_UINT(Tc2_System.MAX_STRING_LENGTH)
) THEN
	expectedStringAsString := 'String with Tc2_System.MAX_STRING_LENGTH characters';
END_IF

messageStringBuilder(
	sFormat := message,
	arg1 := THIS^.AnyToArg(stringToTestAsString),
	arg2 := THIS^.AnyToArg(expectedStringAsString)
);


THIS^.assertorContainer.assertor.assert.strings.unicode.startsWith(
	stringToCheck := stringToTest,
	start := expectedString,
	ignoreCases := TRUE,
	trim := FALSE,
	message			:= ''
);

THIS^.AssertEquals_BOOL(
	Expected 	:= assertionIsWrong,
	Actual 		:= THIS^.assertorContainer.wasAssertionWrong,
	Message 	:= messageStringBuilder.sOut
);

THIS^.AssertEquals_WSTRING(
	Expected 	:= stringToTestBeforeAssertion,
	Actual 		:= stringToTest,
	Message 	:= 'the assertion changed $'stringToTest$''
);

THIS^.AssertEquals_WSTRING(
	Expected 	:= expectedStringBeforeAssertion,
	Actual 		:= expectedString,
	Message 	:= 'the assertion changed $'expectedString$''
);

THIS^.assertorContainer.resetAssertor();

CNM_UnicodeUtilities.NormalizeUtf16String(
	utf16StringBuffer := ADR(stringToTest),
	bufferSize := Tc2_System.MAX_STRING_LENGTH * 2 + 2,
	normalizedStringBuffer := ADR(normalizedStringToTest),
	normalForm := CNM_UnicodeUtilities.NormalizationForm.NFD
);
CNM_UnicodeUtilities.NormalizeUtf16String(
	utf16StringBuffer := ADR(expectedString),
	bufferSize := Tc2_System.MAX_STRING_LENGTH * 2 + 2,
	normalizedStringBuffer := ADR(normalizedExpectedString),
	normalForm := CNM_UnicodeUtilities.NormalizationForm.NFD
);

normalizedUpperStringToTest := normalizedStringToTest;
normalizedUpperExpectedString := normalizedExpectedString;
CNM_UnicodeUtilities.GetUpperCaseUtf16(ADR(normalizedUpperStringToTest));
CNM_UnicodeUtilities.GetUpperCaseUtf16(ADR(normalizedUpperExpectedString));


CNM_UnicodeUtilities.GetUtf16StringLength(
	utf16StringAddress := ADR(normalizedUpperExpectedString),
	characterCount => expectedCharacterCount
);
assertionIsWrong := ((
		CNM_UnicodeUtilities.FindInUtf16String(
			ADR(normalizedUpperStringToTest),
			ADR(normalizedUpperExpectedString),
		) <> 1
	) AND (
		expectedCharacterCount <> 0
	)
);

THIS^.assertorContainer.assertor.assert.strings.unicode.startsWith(
	stringToCheck := stringToTest,
	start := expectedString,
	ignoreCases := TRUE,
	trim		:= FALSE,
	normalizeStrings := TRUE,
	message			:= ''
);

THIS^.AssertEquals_BOOL(
	Expected 	:= assertionIsWrong,
	Actual 		:= THIS^.assertorContainer.wasAssertionWrong,
	Message 	:= messageStringBuilder.sOut
);

THIS^.AssertEquals_WSTRING(
	Expected 	:= stringToTestBeforeAssertion,
	Actual 		:= stringToTest,
	Message 	:= 'the assertion changed $'stringToTest$''
);

THIS^.AssertEquals_WSTRING(
	Expected 	:= expectedStringBeforeAssertion,
	Actual 		:= expectedString,
	Message 	:= 'the assertion changed $'expectedString$''
);
END_METHOD

(*
short summary
==================
This test method tests ``assert.string.unicode.startsWith``
method of CNM_AssertionInterfaces library with various inputs

.. <legal notes>

legal notes
=================
| SPDX-FileCopyrightText: © 2022 ekvip automation GmbH <info@ekvip.de>
| SPDX-License-Identifier: Apache-2.0
| For details check: Apache-2.0_

.. _Apache-2.0: https://www.apache.org/licenses/LICENSE-2.0

.. </legal notes>

*)


METHOD testStartsWithTrim : BOOL
VAR_INPUT
	(* for the test it's the parameter ``stringToCheck`` *)
	stringToTest  	:WSTRING(Tc2_System.MAX_STRING_LENGTH);
	(* for the test it's the parameter ``searchString`` *)
	expectedString	:WSTRING(Tc2_System.MAX_STRING_LENGTH);
END_VAR
VAR 
	(* just the expectation if the assertion to test must be worng or true *)
	assertionIsWrong				:BOOL;
	(* contains the format string for the test message *)
	message							:Tc2_System.T_MaxString;
	(* contains ´´stringToTest´´ trimed *)
	trimedStringToTest				:WSTRING(Tc2_System.MAX_STRING_LENGTH);
	(* contains ´´expectedString´´ trimed *)
	trimedExpectedString			:WSTRING(Tc2_System.MAX_STRING_LENGTH);
	(* used for placeholder string if stringToTest can't be printed *)
	stringToTestAsString 			:Tc2_System.T_MaxString;
	(* used for placeholder string if expectedString can't be printed *)
	expectedStringAsString 			:Tc2_System.T_MaxString;
	(* contains stringToTest in normalized form *)
	normalizedStringToTest			:WSTRING(Tc2_System.MAX_STRING_LENGTH);
	(* contains expectedString in normalized form *)
	normalizedExpectedString		:WSTRING(Tc2_System.MAX_STRING_LENGTH);
	(* contains stringToTest in normalized form trimed *)
	normalizedTrimedStringToTest	:WSTRING(Tc2_System.MAX_STRING_LENGTH);
	(* contains expectedString in normalized form trimed *)
	normalizedTrimedExpectedString	:WSTRING(Tc2_System.MAX_STRING_LENGTH);
	(* holds characterCount of ``expectedString`` *)
	expectedCharacterCount			:UDINT;
	(* TwinCAT printf with the test message *)
	messageStringBuilder			:Tc2_Utilities.FB_FormatString;
	(* hold stringToCheck before assertion *)
	stringToTestBeforeAssertion		:WSTRING(Tc2_System.MAX_STRING_LENGTH);
	(* hold stringToCheck before assertion *)
	expectedStringBeforeAssertion	:WSTRING(Tc2_System.MAX_STRING_LENGTH);
END_VAR
THIS^.assertorContainer.resetAssertor();

stringToTestBeforeAssertion := stringToTest;
expectedStringBeforeAssertion := expectedString;

trimedStringToTest := stringToTest;
trimedExpectedString := expectedString;

// trim the left of both strings
CNM_UnicodeUtilities.TrimLeftUtf16String(ADR(trimedStringToTest));
CNM_UnicodeUtilities.TrimLeftUtf16String(ADR(trimedExpectedString));

CNM_UnicodeUtilities.GetUtf16StringLength(
	utf16StringAddress := ADR(trimedExpectedString),
	characterCount => expectedCharacterCount
);
assertionIsWrong := ((
		CNM_UnicodeUtilities.FindInUtf16String(
			ADR(trimedStringToTest),
			ADR(trimedExpectedString),
		) <> 1
	) AND (
		expectedCharacterCount <> 0
	)
);

message := SEL(
	assertionIsWrong,
	'stringToCheck is $'%s$' start is $'%s$' assertion must be TRUE', 
	'stringToCheck is $'%s$' start is $'%s$' assertion must be FALSE'
);

Tc2_Utilities.WSTRING_TO_STRING2(ADR(stringToTestAsString), ADR(stringToTest), SIZEOF(stringToTestAsString));
Tc2_Utilities.WSTRING_TO_STRING2(ADR(expectedStringAsString), ADR(expectedString), SIZEOF(expectedStringAsString));

IF (
		Tc2_Standard.WLEN(stringToTest) = TO_UINT(Tc2_System.MAX_STRING_LENGTH)
) THEN
	stringToTestAsString := 'String with Tc2_System.MAX_STRING_LENGTH characters';
END_IF
IF (
		Tc2_Standard.WLEN(expectedString) = TO_UINT(Tc2_System.MAX_STRING_LENGTH)
) THEN
	expectedStringAsString := 'String with Tc2_System.MAX_STRING_LENGTH characters';
END_IF

messageStringBuilder(
	sFormat := message,
	arg1 := THIS^.AnyToArg(stringToTestAsString),
	arg2 := THIS^.AnyToArg(expectedStringAsString)
);


THIS^.assertorContainer.assertor.assert.strings.unicode.startsWith(
	stringToCheck := stringToTest,
	start := expectedString,
	ignoreCases := FALSE,
	trim := TRUE,
	normalizeStrings := FALSE,
	message			:= ''
);

THIS^.AssertEquals_BOOL(
	Expected 	:= assertionIsWrong,
	Actual 		:= THIS^.assertorContainer.wasAssertionWrong,
	Message 	:= messageStringBuilder.sOut
);

THIS^.AssertEquals_WSTRING(
	Expected 	:= stringToTestBeforeAssertion,
	Actual 		:= stringToTest,
	Message 	:= 'the assertion changed $'stringToTest$''
);

THIS^.AssertEquals_WSTRING(
	Expected 	:= expectedStringBeforeAssertion,
	Actual 		:= expectedString,
	Message 	:= 'the assertion changed $'expectedString$''
);

THIS^.assertorContainer.resetAssertor();

CNM_UnicodeUtilities.NormalizeUtf16String(
	utf16StringBuffer := ADR(stringToTest),
	bufferSize := Tc2_System.MAX_STRING_LENGTH * 2 + 2,
	normalizedStringBuffer := ADR(normalizedStringToTest),
	normalForm := CNM_UnicodeUtilities.NormalizationForm.NFD
);
CNM_UnicodeUtilities.NormalizeUtf16String(
	utf16StringBuffer := ADR(expectedString),
	bufferSize := Tc2_System.MAX_STRING_LENGTH * 2 + 2,
	normalizedStringBuffer := ADR(normalizedExpectedString),
	normalForm := CNM_UnicodeUtilities.NormalizationForm.NFD
);

normalizedTrimedStringToTest := normalizedStringToTest;
normalizedTrimedExpectedString := normalizedExpectedString;
CNM_UnicodeUtilities.TrimLeftUtf16String(ADR(normalizedTrimedStringToTest));
CNM_UnicodeUtilities.TrimLeftUtf16String(ADR(normalizedTrimedExpectedString));

CNM_UnicodeUtilities.GetUtf16StringLength(
	utf16StringAddress := ADR(normalizedTrimedExpectedString),
	characterCount => expectedCharacterCount
);
assertionIsWrong := ((
		CNM_UnicodeUtilities.FindInUtf16String(
			ADR(normalizedTrimedStringToTest),
			ADR(normalizedTrimedExpectedString),
		) <> 1
	) AND (
		expectedCharacterCount <> 0
	)
);

THIS^.assertorContainer.assertor.assert.strings.unicode.startsWith(
	stringToCheck := stringToTest,
	start := expectedString,
	ignoreCases := FALSE,
	trim		:= TRUE,
	normalizeStrings := TRUE,
	message			:= ''
);

THIS^.AssertEquals_BOOL(
	Expected 	:= assertionIsWrong,
	Actual 		:= THIS^.assertorContainer.wasAssertionWrong,
	Message 	:= messageStringBuilder.sOut
);

THIS^.AssertEquals_WSTRING(
	Expected 	:= stringToTestBeforeAssertion,
	Actual 		:= stringToTest,
	Message 	:= 'the assertion changed $'stringToTest$''
);

THIS^.AssertEquals_WSTRING(
	Expected 	:= expectedStringBeforeAssertion,
	Actual 		:= expectedString,
	Message 	:= 'the assertion changed $'expectedString$''
);
END_METHOD

END_FUNCTION_BLOCK

// ---- AssertionTester/AssertionTests/StringAssertions/classes/UnicodeUtf8StringAssertionTests.TcPOU

(*
short summary
==================
This class tests all methods of Unicode string assertions
with various UTF-8 string combinations as input and checks expected 
outputs are satisfied or not

.. <legal notes>

legal notes
=================
| SPDX-FileCopyrightText: © 2022 ekvip automation GmbH <info@ekvip.de>
| SPDX-License-Identifier: Apache-2.0
| For details check: Apache-2.0_

.. _Apache-2.0: https://www.apache.org/licenses/LICENSE-2.0

.. </legal notes>

methods and properties
======================

*)


FUNCTION_BLOCK UnicodeUtf8StringAssertionTests EXTENDS AbstractAssertorTest
VAR

END_VAR
VAR CONSTANT
	(* prefix to unify the test names *)
	TEST_NAME_PREFIX :STRING := 'assert.string.unicode(utf8).';
END_VAR

THIS^.runIsEmpty();
THIS^.runIsNotEmpty();
THIS^.runContains();
THIS^.runContainsNo();
THIS^.runEndsWith();
THIS^.runStartsWith();
THIS^.runIsEqualTo();
THIS^.runIsNotEqualTo();
THIS^.runLengthIsBetween();
THIS^.runLengthIsExact();
THIS^.runLengthIsMax();
THIS^.runLengthIsMin();

(*

short summary
==================
This test method is a helper function to create a unified test name

.. <legal notes>

legal notes
=================
| SPDX-FileCopyrightText: © 2022 ekvip automation GmbH <info@ekvip.de>
| SPDX-License-Identifier: Apache-2.0
| For details check: Apache-2.0_

.. _Apache-2.0: https://www.apache.org/licenses/LICENSE-2.0

.. </legal notes>

parameters
==========

*)

METHOD PROTECTED getTestNameFor :Tc2_System.T_MaxString
VAR_INPUT
	(* name of the method to test, to create a unified test name *)
	nameOfMethodToTest	:Tc2_System.T_MaxString;
END_VAR
getTestNameFor := Tc2_Standard.CONCAT(THIS^.TEST_NAME_PREFIX, nameOfMethodToTest);
END_METHOD

(*
short summary
==================
This test method tests ``assert.string.unicode.contains``
method of CNM_AssertionInterfaces library with various inputs

.. <legal notes>

legal notes
=================
| SPDX-FileCopyrightText: © 2022 ekvip automation GmbH <info@ekvip.de>
| SPDX-License-Identifier: Apache-2.0
| For details check: Apache-2.0_

.. _Apache-2.0: https://www.apache.org/licenses/LICENSE-2.0

.. </legal notes>

*)


METHOD runContains : BOOL
VAR_INPUT
END_VAR
RETURN (NOT TcUnit.TEST_ORDERED(THIS^.getTestNameFor('contains')));

THIS^.testContains(
	stringToTest := '',
	expectedString := ''
);
THIS^.testContains(
	stringToTest := 'not empty',
	expectedString := ''
);
THIS^.testContains(
	stringToTest := '',
	expectedString := 'not empty'
);
THIS^.testContains(
	stringToTest := 'not empty',
	expectedString := 'not empty'
);
THIS^.testContains(
	stringToTest := '{|}~',
	expectedString := '3649213469328'
);
THIS^.testContains(
	stringToTest := '1one!',
	expectedString := '1'
);
THIS^.testContains(
	stringToTest := '1one!',
	expectedString := 'one'
);
THIS^.testContains(
	stringToTest := '1one!',
	expectedString := '!'
);
THIS^.testContains(
	stringToTest := '$40$n$t$$$"$'',
	expectedString := '$n$t'
);
THIS^.testContains(
	stringToTest := 'frontmiddleback',
	expectedString := 'back'
);
THIS^.testContains(
	stringToTest := 'frontmiddleback',
	expectedString := 'frontmiddlebackfront'
);
THIS^.testContains(
	stringToTest := 'backfrontmiddle',
	expectedString := 'backmiddle'
);
THIS^.testContains(
	stringToTest := 'J;%_iTxQSk?6GfWewt}yMKh1)VXqPA@P1YQ:{EAg:8VJ,/FM;j)xJ[[AvYp/}}SzEgtfYS,1K0.5VtA+VJrB(p#55h2z##mw#F)Y@P6Jz9G@6vb=x#E!cYk(Svr@S*KiPJr1VZ6AjrNback4G=vBJd.E:=,k3!wmuGDe#ZKMD#Vx%?M_0&L0#vT]J,+)ZvU{w%8X0=:XzthmT0VG0QrwpXXCWpFxu6[b!c.BunYYfLQi.,?ut?-{jrC1phTHL)y',
	expectedString := 'J;%_iTxQSk?6GfWewt}yMKh1)VXqPA@P1YQ:{EAg:8VJ,/FM;j)xJ[[AvYp/}}SzEgtfYS,1K0.5VtA+VJrB(p#55h2z##mw#F)Y@P6Jz9G@6vb=x#E!cYk(Svr@S*KiPJr1VZ6AjrNback4G=vBJd.E:=,k3!wmuGDe#ZKMD#Vx%?M_0&L0#vT]J,+)ZvU{w%8X0=:XzthmT0VG0QrwpXXCWpFxu6[b!c.BunYYfLQi.,?ut?-{jrC1phTHL)y'
);
THIS^.testContains(
	stringToTest := 'J;%_iTxQSk?6GfWewt}yMKh1)VXqPA@P1YQ:{EAg:8VJ,/FM;j)xJ[[AvYp/}}SzEgtfYS,1K0.5VtA+VJrB(p#55h2z##mw#F)Y@P6Jz9G@6vb=x#E!cYk(Svr@S*KiPJr1VZ6AjrNback4G=vBJd.E:=,k3!wmuGDe#ZKMD#Vx%?M_0&L0#vT]J,+)ZvU{w%8X0=:XzthmT0VG0QrwpXXCWpFxu6[b!c.BunYYfLQi.,?ut?-{jrC1phTHL)y',
	expectedString := 'J;%_iTxQSk?6GfWewt}yMKh1)VXqPA@P1YQ:{EAg:8VJ,/FM;j)xJ[[AvYp/}}SzEgtfYS,1K0.5VtA+VJrB(p#55h2z##mw#F)Y@P6Jz9G@6vb=x#E!cYk(Svr@S*KiPJr1VZ6AjrNback4G=vBJd.E:=,k3!wmuGDe#ZKMD#Vx%?M_0&L0#vT]J,+)ZvU{w%8X0=:XzthmT0VG0QrwpXXCWpFxu6[b!c.BunYYfLQi.,?ut?-{jrC1phTHL)x'
);
THIS^.testContains(
	stringToTest := UTF8#'∮ E⋅da = Q,  n → ∞, ∑ f(i) = ∏ g(i), ∀x∈ℝ: ⌈x⌉ = −⌊−x⌋, α ∧ ¬β = ¬(¬α ∨ β)',
	expectedString := UTF8#'∑ f(i) = ∏ g(i)'
);
THIS^.testContains(
	stringToTest := UTF8#'ℕ ⊆ ℕ₀ ⊂ ℤ ⊂ ℚ ⊂ ℝ ⊂ ℂ, ⊥ < a ≠ b ≡ c ≤ d ≪ ⊤ ⇒ (A ⇔ B), 2H₂ + O₂ ⇌ 2H₂O, R = 4.7 kΩ, ⌀ 200 mm',
	expectedString := UTF8#'ℕ ⊆ ℕ₀ ⊂ ℤ ⊂ ℚ ⊂ ℝ ⊂ ℂ'
);
THIS^.testContains(
	stringToTest := UTF8#'ℕ ⊆ ℕ₀ ⊂ ℤ ⊂ ℚ ⊂ ℝ ⊂ ℂ, ⊥ < a ≠ b ≡ c ≤ d ≪ ⊤ ⇒ (A ⇔ B), 2H₂ + O₂ ⇌ 2H₂O, R = 4.7 kΩ, ⌀ 200 mm',
	expectedString := UTF8#'ℕ ⊆ ℕ₀ ⊂ ℤ ⊂ ℚ ⊂ ℝ ⊂ ℂ ⇒ (A ⇔ B)'
);
THIS^.testContains(
	stringToTest := UTF8#'ℕ ⊆ ℕ₀ ⊂ ℤ ⊂ ℚ ⊂ ℝ ⊂ ℂ, ⊥ < a ≠ b ≡ c ≤ d ≪ ⊤ ⇒ (A ⇔ B), 2H₂ + O₂ ⇌ 2H₂O, R = 4.7 kΩ, ⌀ 200 mm',
	expectedString := UTF8#'2H₂ + O₂ ⇌ 2H₂O'
);
THIS^.testContains(
	stringToTest := UTF8#'ði ıntəˈnæʃənəl fəˈnɛtık əsoʊsiˈeıʃn Y [ˈʏpsilɔn], Yen [jɛn], Yoga [ˈjoːgɑ]',
	expectedString := UTF8#'ˈnæʃənəl fəˈnɛtık '
);
THIS^.testContains(
	stringToTest := UTF8#'‚‘„“‘’“We’ve been here”´` †, ‡, ‰, •, 3–4, —, −5/+5, ™, …, 1lI|, 0OD, 8B, €',
	expectedString := UTF8#'‚‘„“‘’“We’ve been here”´` †, ‡, ‰, •, 3–4, —, −5/+5, ™, …, 1lI|, 0OD, 8B, €'
);
THIS^.testContains(
	stringToTest := UTF8#'Σὲ γνωρίζω ἀπὸ τὴν κόψη τοῦ σπαθιοῦ τὴν τρομερή,',
	expectedString := UTF8#'τὴν κόψη τοῦ σπαθ'
);
THIS^.testContains(
	stringToTest := UTF8#'გთხოვთ ახლავე გაიაროთ რეგისტრაცია Unicode-ის მეათე საერთაშორისო კონფერენციაზე დასასწრებად',
	expectedString := UTF8#'გაიაროთ რეგისტრაცია Unicode-ის გაიმართება'
);
THIS^.testContains(
	stringToTest := UTF8#'Зарегистрируйтесь сейчас на Десятую Международную Конференцию по Unicode, которая состоится 10-12 марта 1997 года в',
	expectedString := UTF8#'Международную Конференцию по Unicode, которая'
);
THIS^.testContains(
	stringToTest := UTF8#'๏ แผ่นดินฮั่นเสื่อมโทรมแสนสังเวช  พระปกเกศกองบู๊กู้ขึ้นใหม่',
	expectedString := UTF8#'สิบสองกษัตริย์ก่อนหน้าแลถัดไป       สององค์ไซร้โง่เขลาเบาปัญญา  ' 
);
THIS^.testContains(
	stringToTest := UTF8#' ሰማይ አይታረስ ንጉሥ አይከሰስ። ብላ ካለኝ እንደአባቴ በቆመጠኝ።',
	expectedString := UTF8#'አይታረስ ንጉሥ አይከሰስ። ብላ በቆመጠኝ።'
);
THIS^.testContains(
	stringToTest := UTF8#' ᚻᛖ ᚳᚹᚫᚦ ᚦᚫᛏ ᚻᛖ ᛒᚢᛞᛖ ᚩᚾ ᚦᚫᛗ ᛚᚪᚾᛞᛖ ᚾᚩᚱᚦᚹᛖᚪᚱᛞᚢᛗ ᚹᛁᚦ ᚦᚪ ᚹᛖᛥᚫ',
	expectedString := UTF8#'ᚩᚾ ᚦᚫᛗ ᛚᚪᚾᛞᛖ ᚾᚩᚱᚦᚹᛖᚪᚱᛞᚢᛗ ᚹᛁᚦ ᚦᚪ ᚹᛖᛥᚫ'
);
THIS^.testContains(
	stringToTest := UTF8#'⡍⠔⠙⠖ ⡊ ⠙⠕⠝⠰⠞ ⠍⠑⠁⠝ ⠞⠕ ⠎⠁⠹ ⠹⠁⠞ ⡊ ⠅⠝⠪⠂ ⠕⠋ ⠍⠹
  ⠪⠝ ⠅⠝⠪⠇⠫⠛⠑⠂ ⠱⠁⠞ ⠹⠻⠑ ⠊⠎ ⠏⠜⠞⠊⠊⠥⠇⠜⠇⠹ ⠙⠑⠁⠙ ⠁⠃⠳⠞',
	expectedString := UTF8#'⡊ ⠙⠕⠝⠰⠞ ⠍⠑⠁⠝ ⠞⠕ ⠎⠁⠹ ⠹⠁⠞ ⡊ ⠅⠝⠪⠂ ⠕⠋'
);
THIS^.testContains(
	stringToTest := UTF8#'╔══╦══╗  ┌──┬──┐  ╭──┬──╮  ╭──┬──╮  ┏━━┳━━┓  ┎┒┏┑   ╷  ╻ ┏┯┓ ┌┰┐    ▊ ╱╲╱╲╳╳╳',
	expectedString := UTF8#'╦══╗  ┌──┬──┐  ╭──╦══╗'
);
THIS^.testContainsIgnoreCase(
	stringToTest := 'UPPERCASE',
	expectedString := 'CASE'
);
THIS^.testContainsIgnoreCase(
	stringToTest := 'lowercase',
	expectedString := 'case'
);
THIS^.testContainsIgnoreCase(
	stringToTest := 'UPPERCASE',
	expectedString := 'case'
);
THIS^.testContainsIgnoreCase(
	stringToTest := 'lowercase',
	expectedString := 'CASE'
);
THIS^.testContainsIgnoreCase(
	stringToTest := 'lower',
	expectedString := 'UPPER'
);
THIS^.testContainsIgnoreCase(
	stringToTest := UTF8#'UPPERCASE⌷←⍳→⍴∆∇⊃‾⍎⍕⌈',
	expectedString := UTF8#'case⌷←⍳→⍴∆∇⊃‾⍎⍕⌈'
);
THIS^.testContainsIgnoreCase(
	stringToTest := UTF8#'UPPERCASE((V⍳V)=⍳⍴V)/V←,V',
	expectedString := UTF8#'case((V⍳V)=⍳⍴V)/V←'
);

TcUnit.TEST_FINISHED();
END_METHOD

(*
short summary
==================
This test method tests ``assert.string.unicode.containsNo``
method of CNM_AssertionInterfaces library with various inputs

.. <legal notes>

legal notes
=================
| SPDX-FileCopyrightText: © 2022 ekvip automation GmbH <info@ekvip.de>
| SPDX-License-Identifier: Apache-2.0
| For details check: Apache-2.0_

.. _Apache-2.0: https://www.apache.org/licenses/LICENSE-2.0

.. </legal notes>

*)


METHOD runContainsNo : BOOL
RETURN (NOT TcUnit.TEST_ORDERED(THIS^.getTestNameFor('containsNo')));

THIS^.testContainsNo(
	stringToTest := '',
	expectedString := ''
);
THIS^.testContainsNo(
	stringToTest := 'not empty',
	expectedString := ''
);
THIS^.testContainsNo(
	stringToTest := '',
	expectedString := 'not empty'
);
THIS^.testContainsNo(
	stringToTest := 'not empty',
	expectedString := 'not empty'
);
THIS^.testContainsNo(
	stringToTest := '{|}~',
	expectedString := '3649213469328'
);
THIS^.testContainsNo(
	stringToTest := '1one!',
	expectedString := '1'
);
THIS^.testContainsNo(
	stringToTest := '1one!',
	expectedString := 'one'
);
THIS^.testContainsNo(
	stringToTest := '1one!',
	expectedString := '!'
);
THIS^.testContainsNo(
	stringToTest := '$40$n$t$$$"$'',
	expectedString := '$n$t'
);
THIS^.testContainsNo(
	stringToTest := 'frontmiddleback',
	expectedString := 'back'
);
THIS^.testContainsNo(
	stringToTest := 'frontmiddleback',
	expectedString := 'frontmiddlebackfront'
);
THIS^.testContainsNo(
	stringToTest := 'backfrontmiddle',
	expectedString := 'backmiddle'
);
THIS^.testContainsNo(
	stringToTest := 'J;%_iTxQSk?6GfWewt}yMKh1)VXqPA@P1YQ:{EAg:8VJ,/FM;j)xJ[[AvYp/}}SzEgtfYS,1K0.5VtA+VJrB(p#55h2z##mw#F)Y@P6Jz9G@6vb=x#E!cYk(Svr@S*KiPJr1VZ6AjrNback4G=vBJd.E:=,k3!wmuGDe#ZKMD#Vx%?M_0&L0#vT]J,+)ZvU{w%8X0=:XzthmT0VG0QrwpXXCWpFxu6[b!c.BunYYfLQi.,?ut?-{jrC1phTHL)y',
	expectedString := 'J;%_iTxQSk?6GfWewt}yMKh1)VXqPA@P1YQ:{EAg:8VJ,/FM;j)xJ[[AvYp/}}SzEgtfYS,1K0.5VtA+VJrB(p#55h2z##mw#F)Y@P6Jz9G@6vb=x#E!cYk(Svr@S*KiPJr1VZ6AjrNback4G=vBJd.E:=,k3!wmuGDe#ZKMD#Vx%?M_0&L0#vT]J,+)ZvU{w%8X0=:XzthmT0VG0QrwpXXCWpFxu6[b!c.BunYYfLQi.,?ut?-{jrC1phTHL)y'
);
THIS^.testContainsNo(
	stringToTest := 'J;%_iTxQSk?6GfWewt}yMKh1)VXqPA@P1YQ:{EAg:8VJ,/FM;j)xJ[[AvYp/}}SzEgtfYS,1K0.5VtA+VJrB(p#55h2z##mw#F)Y@P6Jz9G@6vb=x#E!cYk(Svr@S*KiPJr1VZ6AjrNback4G=vBJd.E:=,k3!wmuGDe#ZKMD#Vx%?M_0&L0#vT]J,+)ZvU{w%8X0=:XzthmT0VG0QrwpXXCWpFxu6[b!c.BunYYfLQi.,?ut?-{jrC1phTHL)y',
	expectedString := 'J;%_iTxQSk?6GfWewt}yMKh1)VXqPA@P1YQ:{EAg:8VJ,/FM;j)xJ[[AvYp/}}SzEgtfYS,1K0.5VtA+VJrB(p#55h2z##mw#F)Y@P6Jz9G@6vb=x#E!cYk(Svr@S*KiPJr1VZ6AjrNback4G=vBJd.E:=,k3!wmuGDe#ZKMD#Vx%?M_0&L0#vT]J,+)ZvU{w%8X0=:XzthmT0VG0QrwpXXCWpFxu6[b!c.BunYYfLQi.,?ut?-{jrC1phTHL)x'
);
THIS^.testContainsNo(
	stringToTest := UTF8#'∮ E⋅da = Q,  n → ∞, ∑ f(i) = ∏ g(i), ∀x∈ℝ: ⌈x⌉ = −⌊−x⌋, α ∧ ¬β = ¬(¬α ∨ β)',
	expectedString := UTF8#'∑ f(i) = ∏ g(i)'
);
THIS^.testContainsNo(
	stringToTest := UTF8#'ℕ ⊆ ℕ₀ ⊂ ℤ ⊂ ℚ ⊂ ℝ ⊂ ℂ, ⊥ < a ≠ b ≡ c ≤ d ≪ ⊤ ⇒ (A ⇔ B), 2H₂ + O₂ ⇌ 2H₂O, R = 4.7 kΩ, ⌀ 200 mm',
	expectedString := UTF8#'ℕ ⊆ ℕ₀ ⊂ ℤ ⊂ ℚ ⊂ ℝ ⊂ ℂ'
);
THIS^.testContainsNo(
	stringToTest := UTF8#'ℕ ⊆ ℕ₀ ⊂ ℤ ⊂ ℚ ⊂ ℝ ⊂ ℂ, ⊥ < a ≠ b ≡ c ≤ d ≪ ⊤ ⇒ (A ⇔ B), 2H₂ + O₂ ⇌ 2H₂O, R = 4.7 kΩ, ⌀ 200 mm',
	expectedString := UTF8#'ℕ ⊆ ℕ₀ ⊂ ℤ ⊂ ℚ ⊂ ℝ ⊂ ℂ ⇒ (A ⇔ B)'
);
THIS^.testContainsNo(
	stringToTest := UTF8#'ℕ ⊆ ℕ₀ ⊂ ℤ ⊂ ℚ ⊂ ℝ ⊂ ℂ, ⊥ < a ≠ b ≡ c ≤ d ≪ ⊤ ⇒ (A ⇔ B), 2H₂ + O₂ ⇌ 2H₂O, R = 4.7 kΩ, ⌀ 200 mm',
	expectedString := UTF8#'2H₂ + O₂ ⇌ 2H₂O'
);
THIS^.testContainsNo(
	stringToTest := UTF8#'ði ıntəˈnæʃənəl fəˈnɛtık əsoʊsiˈeıʃn Y [ˈʏpsilɔn], Yen [jɛn], Yoga [ˈjoːgɑ]',
	expectedString := UTF8#'ˈnæʃənəl fəˈnɛtık '
);
THIS^.testContainsNo(
	stringToTest := UTF8#'‚‘„“‘’“We’ve been here”´` †, ‡, ‰, •, 3–4, —, −5/+5, ™, …, 1lI|, 0OD, 8B, €',
	expectedString := UTF8#'‚‘„“‘’“We’ve been here”´` †, ‡, ‰, •, 3–4, —, −5/+5, ™, …, 1lI|, 0OD, 8B, €'
);
THIS^.testContainsNo(
	stringToTest := UTF8#'Σὲ γνωρίζω ἀπὸ τὴν κόψη τοῦ σπαθιοῦ τὴν τρομερή,',
	expectedString := UTF8#'τὴν κόψη τοῦ σπαθ'
);
THIS^.testContainsNo(
	stringToTest := UTF8#'გთხოვთ ახლავე გაიაროთ რეგისტრაცია Unicode-ის მეათე საერთაშორისო კონფერენციაზე დასასწრებად',
	expectedString := UTF8#'გაიაროთ რეგისტრაცია Unicode-ის გაიმართება'
);
THIS^.testContainsNo(
	stringToTest := UTF8#'Зарегистрируйтесь сейчас на Десятую Международную Конференцию по Unicode, которая состоится 10-12 марта 1997 года в',
	expectedString := UTF8#'Международную Конференцию по Unicode, которая'
);
THIS^.testContainsNo(
	stringToTest := UTF8#'๏ แผ่นดินฮั่นเสื่อมโทรมแสนสังเวช  พระปกเกศกองบู๊กู้ขึ้นใหม่',
	expectedString := UTF8#'สิบสองกษัตริย์ก่อนหน้าแลถัดไป       สององค์ไซร้โง่เขลาเบาปัญญา  ' 
);
THIS^.testContainsNo(
	stringToTest := UTF8#' ሰማይ አይታረስ ንጉሥ አይከሰስ። ብላ ካለኝ እንደአባቴ በቆመጠኝ።',
	expectedString := UTF8#'አይታረስ ንጉሥ አይከሰስ። ብላ በቆመጠኝ።'
);
THIS^.testContainsNo(
	stringToTest := UTF8#' ᚻᛖ ᚳᚹᚫᚦ ᚦᚫᛏ ᚻᛖ ᛒᚢᛞᛖ ᚩᚾ ᚦᚫᛗ ᛚᚪᚾᛞᛖ ᚾᚩᚱᚦᚹᛖᚪᚱᛞᚢᛗ ᚹᛁᚦ ᚦᚪ ᚹᛖᛥᚫ',
	expectedString := UTF8#'ᚩᚾ ᚦᚫᛗ ᛚᚪᚾᛞᛖ ᚾᚩᚱᚦᚹᛖᚪᚱᛞᚢᛗ ᚹᛁᚦ ᚦᚪ ᚹᛖᛥᚫ'
);
THIS^.testContainsNo(
	stringToTest := UTF8#'⡍⠔⠙⠖ ⡊ ⠙⠕⠝⠰⠞ ⠍⠑⠁⠝ ⠞⠕ ⠎⠁⠹ ⠹⠁⠞ ⡊ ⠅⠝⠪⠂ ⠕⠋ ⠍⠹
  ⠪⠝ ⠅⠝⠪⠇⠫⠛⠑⠂ ⠱⠁⠞ ⠹⠻⠑ ⠊⠎ ⠏⠜⠞⠊⠊⠥⠇⠜⠇⠹ ⠙⠑⠁⠙ ⠁⠃⠳⠞',
	expectedString := UTF8#'⡊ ⠙⠕⠝⠰⠞ ⠍⠑⠁⠝ ⠞⠕ ⠎⠁⠹ ⠹⠁⠞ ⡊ ⠅⠝⠪⠂ ⠕⠋'
);
THIS^.testContainsNo(
	stringToTest := UTF8#'╔══╦══╗  ┌──┬──┐  ╭──┬──╮  ╭──┬──╮  ┏━━┳━━┓  ┎┒┏┑   ╷  ╻ ┏┯┓ ┌┰┐    ▊ ╱╲╱╲╳╳╳',
	expectedString := UTF8#'╦══╗  ┌──┬──┐  ╭──╦══╗'
);

THIS^.testContainsNoIgnoreCase(
	stringToTest := 'UPPERCASE',
	expectedString := 'CASE'
);
THIS^.testContainsNoIgnoreCase(
	stringToTest := 'lowercase',
	expectedString := 'case'
);
THIS^.testContainsNoIgnoreCase(
	stringToTest := 'UPPERCASE',
	expectedString := 'case'
);
THIS^.testContainsNoIgnoreCase(
	stringToTest := 'lowercase',
	expectedString := 'CASE'
);
THIS^.testContainsNoIgnoreCase(
	stringToTest := 'lower',
	expectedString := 'UPPER'
);
THIS^.testContainsNoIgnoreCase(
	stringToTest := UTF8#'UPPERCASE⌷←⍳→⍴∆∇⊃‾⍎⍕⌈',
	expectedString := UTF8#'case⌷←⍳→⍴∆∇⊃‾⍎⍕⌈'
);
THIS^.testContainsNoIgnoreCase(
	stringToTest := UTF8#'UPPERCASE((V⍳V)=⍳⍴V)/V←,V',
	expectedString := UTF8#'case((V⍳V)=⍳⍴V)/V←'
);

TcUnit.TEST_FINISHED();
END_METHOD

(*
short summary
==================
This test method tests ``assert.string.unicode.endsWith``
method of CNM_AssertionInterfaces library with various inputs

.. <legal notes>

legal notes
=================
| SPDX-FileCopyrightText: © 2022 ekvip automation GmbH <info@ekvip.de>
| SPDX-License-Identifier: Apache-2.0
| For details check: Apache-2.0_

.. _Apache-2.0: https://www.apache.org/licenses/LICENSE-2.0

.. </legal notes>

*)


METHOD runEndsWith : BOOL
VAR_INPUT
END_VAR
RETURN (NOT TcUnit.TEST_ORDERED(THIS^.getTestNameFor('endsWith')));

THIS^.testEndsWith(
	stringToTest := '',
	expectedString := ''
);
THIS^.testEndsWith(
	stringToTest := 'not empty',
	expectedString := ''
);
THIS^.testEndsWith(
	stringToTest := '',
	expectedString := 'not empty'
);
THIS^.testEndsWith(
	stringToTest := 'not empty',
	expectedString := 'not empty'
);
THIS^.testEndsWith(
	stringToTest := '{|}~',
	expectedString := '3649213469328'
);
THIS^.testEndsWith(
	stringToTest := '1one!',
	expectedString := '1'
);
THIS^.testEndsWith(
	stringToTest := '1one!',
	expectedString := 'one'
);
THIS^.testEndsWith(
	stringToTest := '1one!',
	expectedString := '!'
);
THIS^.testEndsWith(
	stringToTest := '$40$n$t$$$"$'',
	expectedString := '$n$t'
);
THIS^.testEndsWith(
	stringToTest := '$40$$$"$'$n$t',
	expectedString := '$n$t'
);
THIS^.testEndsWith(
	stringToTest := 'frontmiddleback',
	expectedString := 'back'
);
THIS^.testEndsWith(
	stringToTest := 'frontmiddleback',
	expectedString := 'frontmiddlebackfront'
);
THIS^.testEndsWith(
	stringToTest := 'backfrontmiddle',
	expectedString := 'backmiddle'
);
THIS^.testEndsWith(
	stringToTest := 'J;%_iTxQSk?6GfWewt}yMKh1)VXqPA@P1YQ:{EAg:8VJ,/FM;j)xJ[[AvYp/}}SzEgtfYS,1K0.5VtA+VJrB(p#55h2z##mw#F)Y@P6Jz9G@6vb=x#E!cYk(Svr@S*KiPJr1VZ6AjrNback4G=vBJd.E:=,k3!wmuGDe#ZKMD#Vx%?M_0&L0#vT]J,+)ZvU{w%8X0=:XzthmT0VG0QrwpXXCWpFxu6[b!c.BunYYfLQi.,?ut?-{jrC1phTHL)y',
	expectedString := 'J;%_iTxQSk?6GfWewt}yMKh1)VXqPA@P1YQ:{EAg:8VJ,/FM;j)xJ[[AvYp/}}SzEgtfYS,1K0.5VtA+VJrB(p#55h2z##mw#F)Y@P6Jz9G@6vb=x#E!cYk(Svr@S*KiPJr1VZ6AjrNback4G=vBJd.E:=,k3!wmuGDe#ZKMD#Vx%?M_0&L0#vT]J,+)ZvU{w%8X0=:XzthmT0VG0QrwpXXCWpFxu6[b!c.BunYYfLQi.,?ut?-{jrC1phTHL)y'
);
THIS^.testEndsWith(
	stringToTest := 'J;%_iTxQSk?6GfWewt}yMKh1)VXqPA@P1YQ:{EAg:8VJ,/FM;j)xJ[[AvYp/}}SzEgtfYS,1K0.5VtA+VJrB(p#55h2z##mw#F)Y@P6Jz9G@6vb=x#E!cYk(Svr@S*KiPJr1VZ6AjrNback4G=vBJd.E:=,k3!wmuGDe#ZKMD#Vx%?M_0&L0#vT]J,+)ZvU{w%8X0=:XzthmT0VG0QrwpXXCWpFxu6[b!c.BunYYfLQi.,?ut?-{jrC1phTHL)y',
	expectedString := 'J;%_iTxQSk?6GfWewt}yMKh1)VXqPA@P1YQ:{EAg:8VJ,/FM;j)xJ[[AvYp/}}SzEgtfYS,1K0.5VtA+VJrB(p#55h2z##mw#F)Y@P6Jz9G@6vb=x#E!cYk(Svr@S*KiPJr1VZ6AjrNback4G=vBJd.E:=,k3!wmuGDe#ZKMD#Vx%?M_0&L0#vT]J,+)ZvU{w%8X0=:XzthmT0VG0QrwpXXCWpFxu6[b!c.BunYYfLQi.,?ut?-{jrC1phTHL)x'
);
THIS^.testEndsWith(
	stringToTest := UTF8#'∮ E⋅da = Q,  n → ∞, ∑ f(i) = ∏ g(i), ∀x∈ℝ: ⌈x⌉ = −⌊−x⌋, α ∧ ¬β = ¬(¬α ∨ β)',
	expectedString := UTF8#'α ∧ ¬β = ¬(¬α ∨ β)'
);
THIS^.testEndsWith(
	stringToTest := UTF8#'ℕ ⊆ ℕ₀ ⊂ ℤ ⊂ ℚ ⊂ ℝ ⊂ ℂ, ⊥ < a ≠ b ≡ c ≤ d ≪ ⊤ ⇒ (A ⇔ B), 2H₂ + O₂ ⇌ 2H₂O, R = 4.7 kΩ, ⌀ 200 mm',
	expectedString := UTF8#'2H₂ + O₂ ⇌ 2H₂O, R = 4.7 kΩ, ⌀ 200 mm'
);
THIS^.testEndsWith(
	stringToTest := UTF8#'ℕ ⊆ ℕ₀ ⊂ ℤ ⊂ ℚ ⊂ ℝ ⊂ ℂ, ⊥ < a ≠ b ≡ c ≤ d ≪ ⊤ ⇒ (A ⇔ B), 2H₂ + O₂ ⇌ 2H₂O, R = 4.7 kΩ, ⌀ 200 mm',
	expectedString := UTF8#'2H₂ + O₂ ⇌ 2H₂O, R = 4.7 kΩ, ⌀ 200 mm ℕ ⊆ ℕ₀ ⊂ ℤ ⊂ ℚ ⊂ ℝ ⊂ ℂ ⇒ (A ⇔ B)'
);
THIS^.testEndsWith(
	stringToTest := UTF8#'ℕ ⊆ ℕ₀ ⊂ ℤ ⊂ ℚ ⊂ ℝ ⊂ ℂ, ⊥ < a ≠ b ≡ c ≤ d ≪ ⊤ ⇒ (A ⇔ B), 2H₂ + O₂ ⇌ 2H₂O, R = 4.7 kΩ, ⌀ 200 mm',
	expectedString := UTF8#'2H₂ + O₂ ⇌ 2H₂O'
);
THIS^.testEndsWith(
	stringToTest := UTF8#'ði ıntəˈnæʃənəl fəˈnɛtık əsoʊsiˈeıʃn Y [ˈʏpsilɔn], Yen [jɛn], Yoga [ˈjoːgɑ]ˈnæʃənəl fəˈnɛtık ',
	expectedString := UTF8#'ˈnæʃənəl fəˈnɛtık '
);
THIS^.testEndsWith(
	stringToTest := UTF8#'‚‘„“‘’“We’ve been here”´` †, ‡, ‰, •, 3–4, —, −5/+5, ™, …, 1lI|, 0OD, 8B, €',
	expectedString := UTF8#'‚‘„“‘’“We’ve been here”´` †, ‡, ‰, •, 3–4, —, −5/+5, ™, …, 1lI|, 0OD, 8B, €'
);
THIS^.testEndsWith(
	stringToTest := UTF8#'Σὲ γνωρίζω ἀπὸ τὴν κόψη τοῦ σπαθιοῦ τὴν τρομερή,',
	expectedString := UTF8#'τὴν κόψη τοῦ σπαθ'
);
THIS^.testEndsWith(
	stringToTest := UTF8#'გთხოვთ ახლავე გაიაროთ რეგისტრაცია Unicode-ის მეათე საერთაშორისო კონფერენციაზე დასასწრებად',
	expectedString := UTF8#'რომელიც გაიმართება'
);
THIS^.testEndsWith(
	stringToTest := UTF8#'Зарегистрируйтесь сейчас на Десятую Международную Конференцию по Unicode, которая состоится 10-12 марта 1997 года в',
	expectedString := UTF8#'Международную Конференцию по Unicode, которая'
);
THIS^.testEndsWith(
	stringToTest := UTF8#'๏ แผ่นดินฮั่นเสื่อมโทรมแสนสังเวช  พระปกเกศกองบู๊กู้ขึ้นใหม่',
	expectedString := UTF8#'สิบสองกษัตริย์ก่อนหน้าแลถัดไป       สององค์ไซร้โง่เขลาเบาปัญญา ' 
);
THIS^.testEndsWith(
	stringToTest := UTF8#' ሰማይ አይታረስ ንጉሥ አይከሰስ። ብላ ካለኝ እንደአባቴ በቆመጠኝ።',
	expectedString := UTF8#'አይታረስ ንጉሥ አይከሰስ። በቆመጠኝ።'
);
THIS^.testEndsWith(
	stringToTest := UTF8#' ᚻᛖ ᚳᚹᚫᚦ ᚦᚫᛏ ᚻᛖ ᛒᚢᛞᛖ ᚩᚾ ᚦᚫᛗ ᛚᚪᚾᛞᛖ ᚾᚩᚱᚦᚹᛖᚪᚱᛞᚢᛗ ᚹᛁᚦ ᚦᚪ ᚹᛖᛥᚫ',
	expectedString := UTF8#'ᚩᚾ ᚦᚫᛗ ᛚᚪᚾᛞᛖ ᚾᚩᚱᚦᚹᛖᚪᚱᛞᚢᛗ ᚹᛁᚦ ᚦᚪ ᚹᛖᛥᚫ'
);
THIS^.testEndsWith(
	stringToTest := UTF8#'⡍⠔⠙⠖ ⡊ ⠙⠕⠝⠰⠞ ⠍⠑⠁⠝ ⠞⠕ ⠎⠁⠹ ⠹⠁⠞ ⡊ ⠅⠝⠪⠂ ⠕⠋ ⠍⠹
  ⠪⠝ ⠅⠝⠪⠇⠫⠛⠑⠂ ⠱⠁⠞ ⠹⠻⠑ ⠊⠎ ⠏⠜⠞⠊⠊⠥⠇⠜⠇⠹ ⠙⠑⠁⠙ ⠁⠃⠳⠞',
	expectedString := UTF8#'⠱⠁⠞ ⠹⠻⠑ ⠊⠎ ⠏⠜⠞⠊⠊⠥⠇⠜⠇⠹ ⠙'
);
THIS^.testEndsWith(
	stringToTest := UTF8#'╔══╦══╗  ┌──┬──┐  ╭──┬──╮  ╭──┬──╮  ┏━━┳━━┓  ┎┒┏┑   ╷  ╻ ┏┯┓ ┌┰┐    ▊ ╱╲╱╲╳╳╳',
	expectedString := UTF8#'┎┒┏┑   ╷  ╻ ┏┯┓ ┌┰┐    ▊ ╱╲╱╲╳╳╳'
);

THIS^.testEndsWithIgnoreCase(
	stringToTest := 'UPPERCASE',
	expectedString := 'CASE'
);
THIS^.testEndsWithIgnoreCase(
	stringToTest := 'lowercase',
	expectedString := 'case'
);
THIS^.testEndsWithIgnoreCase(
	stringToTest := 'UPPERCASE',
	expectedString := 'case'
);
THIS^.testEndsWithIgnoreCase(
	stringToTest := 'lowercase',
	expectedString := 'CASE'
);
THIS^.testEndsWithIgnoreCase(
	stringToTest := 'lower',
	expectedString := 'UPPER'
);
THIS^.testEndsWithIgnoreCase(
	stringToTest := UTF8#'UPPERCASE⌷←⍳→⍴∆∇⊃‾⍎⍕⌈',
	expectedString := UTF8#'case⌷←⍳→⍴∆∇⊃‾⍎⍕⌈'
);
THIS^.testEndsWithIgnoreCase(
	stringToTest := UTF8#'UPPERCASE((V⍳V)=⍳⍴V)/V←,V',
	expectedString := UTF8#'case((V⍳V)=⍳⍴V)/V←'
);

THIS^.testEndsWithTrim(
	stringToTest := 'frontmiddleback$t',
	expectedString := 'back'
);
THIS^.testEndsWithTrim(
	stringToTest := 'frontmiddleback',
	expectedString := 'back$t'
);
THIS^.testEndsWithTrim(
	stringToTest := 'frontmiddleback$20',
	expectedString := 'back'
);
THIS^.testEndsWithTrim(
	stringToTest := 'frontmiddleback',
	expectedString := 'back$20'
);
THIS^.testEndsWithTrim(
	stringToTest := 'frontmiddleback$t$n$r$p$l',
	expectedString := 'back$r$t$n$l$p$20'
);
THIS^.testEndsWithTrim(
	stringToTest := 'frontmiddleback$t$n$r$p$l',
	expectedString := 'back$t$n$r$p$l$20'
);
THIS^.testEndsWithTrim(
	stringToTest := UTF8#'frontmiddleback⌷←⍳→⍴∆∇⊃‾⍎$t$n$r$p$l',
	expectedString := UTF8#'back⌷←⍳→⍴∆∇⊃‾⍎'
);
THIS^.testEndsWithTrim(
	stringToTest := UTF8#'frontmiddleback⌷←⍳→⍴∆∇⊃‾⍎$t$n$r$p$l',
	expectedString := UTF8#'back⌷→⍴∆∇⊃‾⍎'
);

TcUnit.TEST_FINISHED();
END_METHOD

(*
short summary
==================
This test method tests ``assert.string.unicode.IsEmpty``
method of CNM_AssertionInterfaces library with various inputs

.. <legal notes>

legal notes
=================
| SPDX-FileCopyrightText: © 2022 ekvip automation GmbH <info@ekvip.de>
| SPDX-License-Identifier: Apache-2.0
| For details check: Apache-2.0_

.. _Apache-2.0: https://www.apache.org/licenses/LICENSE-2.0

.. </legal notes>

*)


METHOD runIsEmpty : BOOL
VAR_INPUT
END_VAR
RETURN (NOT TcUnit.TEST_ORDERED(THIS^.getTestNameFor('IsEmpty')));

THIS^.testIsEmpty(
	stringToTest := ''
);
THIS^.testIsEmpty(
	stringToTest := 'not empty'
);
THIS^.testIsEmpty(
	stringToTest := '{|}~'
);
THIS^.testIsEmpty(
	stringToTest := '3649213469328'
);
THIS^.testIsEmpty(
	stringToTest := '1one!'
);
THIS^.testIsEmpty(
	stringToTest := '$40$n$t$$$"$''
);
THIS^.testIsEmpty(
	stringToTest := '$n$t'
);
THIS^.testIsEmpty(
	stringToTest := 'frontmiddleback'
);
THIS^.testIsEmpty(
	stringToTest := 'backfrontmiddle'
);
THIS^.testIsEmpty(
	stringToTest := 'J;%_iTxQSk?6GfWewt}yMKh1)VXqPA@P1YQ:{EAg:8VJ,/FM;j)xJ[[AvYp/}}SzEgtfYS,1K0.5VtA+VJrB(p#55h2z##mw#F)Y@P6Jz9G@6vb=x#E!cYk(Svr@S*KiPJr1VZ6AjrNback4G=vBJd.E:=,k3!wmuGDe#ZKMD#Vx%?M_0&L0#vT]J,+)ZvU{w%8X0=:XzthmT0VG0QrwpXXCWpFxu6[b!c.BunYYfLQi.,?ut?-{jrC1phTHL)y'
);
THIS^.testIsEmpty(
	stringToTest := UTF8#'∮ E⋅da = Q,  n → ∞, ∑ f(i) = ∏ g(i), ∀x∈ℝ: ⌈x⌉ = −⌊−x⌋, α ∧ ¬β = ¬(¬α ∨ β)',
);
THIS^.testIsEmpty(
	stringToTest := UTF8#'ℕ ⊆ ℕ₀ ⊂ ℤ ⊂ ℚ ⊂ ℝ ⊂ ℂ, ⊥ < a ≠ b ≡ c ≤ d ≪ ⊤ ⇒ (A ⇔ B), 2H₂ + O₂ ⇌ 2H₂O, R = 4.7 kΩ, ⌀ 200 mm',
);
THIS^.testIsEmpty(
	stringToTest := UTF8#'ði ıntəˈnæʃənəl fəˈnɛtık əsoʊsiˈeıʃn Y [ˈʏpsilɔn], Yen [jɛn], Yoga [ˈjoːgɑ]',
);
THIS^.testIsEmpty(
	stringToTest := UTF8#'‚‘„“‘’“We’ve been here”´` †, ‡, ‰, •, 3–4, —, −5/+5, ™, …, 1lI|, 0OD, 8B, €',
);
THIS^.testIsEmpty(
	stringToTest := UTF8#'Σὲ γνωρίζω ἀπὸ τὴν κόψη τοῦ σπαθιοῦ τὴν τρομερή,',
);
THIS^.testIsEmpty(
	stringToTest := UTF8#'გთხოვთ ახლავე გაიაროთ რეგისტრაცია Unicode-ის მეათე საერთაშორისო კონფერენციაზე დასასწრებად',
);
THIS^.testIsEmpty(
	stringToTest := UTF8#'Зарегистрируйтесь сейчас на Десятую Международную Конференцию по Unicode, которая состоится 10-12 марта 1997 года в',
);
THIS^.testIsEmpty(
	stringToTest := UTF8#'๏ แผ่นดินฮั่นเสื่อมโทรมแสนสังเวช  พระปกเกศกองบู๊กู้ขึ้นใหม่',
);
THIS^.testIsEmpty(
	stringToTest := UTF8#' ሰማይ አይታረስ ንጉሥ አይከሰስ። ብላ ካለኝ እንደአባቴ በቆመጠኝ።',
);
THIS^.testIsEmpty(
	stringToTest := UTF8#' ᚻᛖ ᚳᚹᚫᚦ ᚦᚫᛏ ᚻᛖ ᛒᚢᛞᛖ ᚩᚾ ᚦᚫᛗ ᛚᚪᚾᛞᛖ ᚾᚩᚱᚦᚹᛖᚪᚱᛞᚢᛗ ᚹᛁᚦ ᚦᚪ ᚹᛖᛥᚫ',
);
THIS^.testIsEmpty(
	stringToTest := UTF8#'⡍⠔⠙⠖ ⡊ ⠙⠕⠝⠰⠞ ⠍⠑⠁⠝ ⠞⠕ ⠎⠁⠹ ⠹⠁⠞ ⡊ ⠅⠝⠪⠂ ⠕⠋ ⠍⠹
  ⠪⠝ ⠅⠝⠪⠇⠫⠛⠑⠂ ⠱⠁⠞ ⠹⠻⠑ ⠊⠎ ⠏⠜⠞⠊⠊⠥⠇⠜⠇⠹ ⠙⠑⠁⠙ ⠁⠃⠳⠞',
);
THIS^.testIsEmpty(
	stringToTest := UTF8#'╔══╦══╗  ┌──┬──┐  ╭──┬──╮  ╭──┬──╮  ┏━━┳━━┓  ┎┒┏┑   ╷  ╻ ┏┯┓ ┌┰┐    ▊ ╱╲╱╲╳╳╳',
);

TcUnit.TEST_FINISHED();
END_METHOD

(*
short summary
==================
This test method tests ``assert.string.unicode.isEqualTo``
method of CNM_AssertionInterfaces library with various inputs

.. <legal notes>

legal notes
=================
| SPDX-FileCopyrightText: © 2022 ekvip automation GmbH <info@ekvip.de>
| SPDX-License-Identifier: Apache-2.0
| For details check: Apache-2.0_

.. _Apache-2.0: https://www.apache.org/licenses/LICENSE-2.0

.. </legal notes>

*)


METHOD runIsEqualTo : BOOL
VAR_INPUT
END_VAR
RETURN (NOT TcUnit.TEST_ORDERED(THIS^.getTestNameFor('isEqualTo')));

THIS^.testisEqualTo(
	stringToTest := '',
	expectedString := ''
);
THIS^.testisEqualTo(
	stringToTest := 'not empty',
	expectedString := ''
);
THIS^.testisEqualTo(
	stringToTest := '',
	expectedString := 'not empty'
);
THIS^.testisEqualTo(
	stringToTest := 'not empty',
	expectedString := 'not'
);
THIS^.testisEqualTo(
	stringToTest := 'not empty',
	expectedString := 'not empty'
);
THIS^.testisEqualTo(
	stringToTest := '{|}~',
	expectedString := '3649213469328'
);
THIS^.testisEqualTo(
	stringToTest := '1one!',
	expectedString := '1one'
);
THIS^.testisEqualTo(
	stringToTest := '1one!',
	expectedString := '1one!'
);

THIS^.testisEqualTo(
	stringToTest := '$40$n$t$$$"$'',
	expectedString := '$n$t'
);
THIS^.testisEqualTo(
	stringToTest := '$40$n$t$$$"$'',
	expectedString := '$40$n$t$$$"$''
);
THIS^.testisEqualTo(
	stringToTest := 'frontmiddleback',
	expectedString := 'back'
);
THIS^.testisEqualTo(
	stringToTest := 'frontmiddleback',
	expectedString := 'frontmiddlebackfront'
);
THIS^.testisEqualTo(
	stringToTest := 'backfrontmiddle',
	expectedString := 'backmiddle'
);
THIS^.testisEqualTo(
	stringToTest := 'J;%_iTxQSk?6GfWewt}yMKh1)VXqPA@P1YQ:{EAg:8VJ,/FM;j)xJ[[AvYp/}}SzEgtfYS,1K0.5VtA+VJrB(p#55h2z##mw#F)Y@P6Jz9G@6vb=x#E!cYk(Svr@S*KiPJr1VZ6AjrNback4G=vBJd.E:=,k3!wmuGDe#ZKMD#Vx%?M_0&L0#vT]J,+)ZvU{w%8X0=:XzthmT0VG0QrwpXXCWpFxu6[b!c.BunYYfLQi.,?ut?-{jrC1phTHL)y',
	expectedString := 'J;%_iTxQSk?6GfWewt}yMKh1)VXqPA@P1YQ:{EAg:8VJ,/FM;j)xJ[[AvYp/}}SzEgtfYS,1K0.5VtA+VJrB(p#55h2z##mw#F)Y@P6Jz9G@6vb=x#E!cYk(Svr@S*KiPJr1VZ6AjrNback4G=vBJd.E:=,k3!wmuGDe#ZKMD#Vx%?M_0&L0#vT]J,+)ZvU{w%8X0=:XzthmT0VG0QrwpXXCWpFxu6[b!c.BunYYfLQi.,?ut?-{jrC1phTHL)y'
);
THIS^.testisEqualTo(
	stringToTest := 'J;%_iTxQSk?6GfWewt}yMKh1)VXqPA@P1YQ:{EAg:8VJ,/FM;j)xJ[[AvYp/}}SzEgtfYS,1K0.5VtA+VJrB(p#55h2z##mw#F)Y@P6Jz9G@6vb=x#E!cYk(Svr@S*KiPJr1VZ6AjrNback4G=vBJd.E:=,k3!wmuGDe#ZKMD#Vx%?M_0&L0#vT]J,+)ZvU{w%8X0=:XzthmT0VG0QrwpXXCWpFxu6[b!c.BunYYfLQi.,?ut?-{jrC1phTHL)y',
	expectedString := 'J;%_iTxQSk?6GfWewt}yMKh1)VXqPA@P1YQ:{EAg:8VJ,/FM;j)xJ[[AvYp/}}SzEgtfYS,1K0.5VtA+VJrB(p#55h2z##mw#F)Y@P6Jz9G@6vb=x#E!cYk(Svr@S*KiPJr1VZ6AjrNback4G=vBJd.E:=,k3!wmuGDe#ZKMD#Vx%?M_0&L0#vT]J,+)ZvU{w%8X0=:XzthmT0VG0QrwpXXCWpFxu6[b!c.BunYYfLQi.,?ut?-{jrC1phTHL)x'
);
THIS^.testisEqualTo(
	stringToTest := UTF8#'∮ E⋅da = Q,  n → ∞, ∑ f(i) = ∏ g(i), ∀x∈ℝ: ⌈x⌉ = −⌊−x⌋, α ∧ ¬β = ¬(¬α ∨ β)',
	expectedString := UTF8#'∮ E⋅da = Q,  n → ∞, ∑ f(i) = ∏ g(i), ∀x∈ℝ: ⌈x⌉ = −⌊−x⌋, α ∧ ¬β = ¬(¬α ∨ β)'
);
THIS^.testisEqualTo(
	stringToTest := UTF8#'ℕ ⊆ ℕ₀ ⊂ ℤ ⊂ ℚ ⊂ ℝ ⊂ ℂ, ⊥ < a ≠ b ≡ c ≤ d ≪ ⊤ ⇒ (A ⇔ B), 2H₂ + O₂ ⇌ 2H₂O, R = 4.7 kΩ, ⌀ 200 mm',
	expectedString := UTF8#'ℕ ⊆ ℕ₀ ⊂ ℤ ⊂ ℚ ⊂ ℝ ⊂ ℂ'
);
THIS^.testisEqualTo(
	stringToTest := UTF8#'ℕ ⊆ ℕ₀ ⊂ ℤ ⊂ ℚ ⊂ ℝ ⊂ ℂ, ⊥ < a ≠ b ≡ c ≤ d ≪ ⊤ ⇒ (A ⇔ B), 2H₂ + O₂ ⇌ 2H₂O, R = 4.7 kΩ, ⌀ 200 mm',
	expectedString := UTF8#'ℕ ⊆ ℕ₀ ⊂ ℤ ⊂ ℚ ⊂ ℝ ⊂ ℂ, ⊥ < a ≠ b ≡ c ≤ d ≪ ⊤ ⇒ (A ⇔ B), 2H₂ + O₂ ⇌ 2H₂O, R = 4.7 kΩ, ⌀ 200 mm'
);
THIS^.testisEqualTo(
	stringToTest := UTF8#'ði ıntəˈnæʃənəl fəˈnɛtık əsoʊsiˈeıʃn Y [ˈʏpsilɔn], Yen [jɛn], Yoga [ˈjoːgɑ]',
	expectedString := UTF8#'ˈnæʃənəl fəˈnɛtık '
);
THIS^.testisEqualTo(
	stringToTest := UTF8#'‚‘„“‘’“We’ve been here”´` †, ‡, ‰, •, 3–4, —, −5/+5, ™, …, 1lI|, 0OD, 8B, €',
	expectedString := UTF8#'‚‘„“‘’“We’ve been here”´` †, ‡, ‰, •, 3–4, —, −5/+5, ™, …, 1lI|, 0OD, 8B, €'
);
THIS^.testisEqualTo(
	stringToTest := UTF8#'Σὲ γνωρίζω ἀπὸ τὴν κόψη τοῦ σπαθιοῦ τὴν τρομερή,',
	expectedString := UTF8#'τὴν κόψη τοῦ σπαθ'
);
THIS^.testisEqualTo(
	stringToTest := UTF8#'გთხოვთ ახლავე გაიაროთ რეგისტრაცია Unicode-ის მეათე საერთაშორისო კონფერენციაზე დასასწრებად',
	expectedString := UTF8#'გთხოვთ ახლავე გაიაროთ რეგისტრაცია Unicode-ის მეათე საერთაშორისო კონფერენციაზე დასასწრებად'
);
THIS^.testisEqualTo(
	stringToTest := UTF8#'Зарегистрируйтесь сейчас на Десятую Международную Конференцию по Unicode, которая состоится 10-12 марта 1997 года в',
	expectedString := UTF8#'Международную Конференцию по Unicode, которая'
);
THIS^.testisEqualTo(
	stringToTest := UTF8#'๏ แผ่นดินฮั่นเสื่อมโทรมแสนสังเวช  พระปกเกศกองบู๊กู้ขึ้นใหม่',
	expectedString := UTF8#'๏ แผ่นดินฮั่นเสื่อมโทรมแสนสังเวช  พระปกเกศกองบู๊กู้ขึ้นใหม่'
);
THIS^.testisEqualTo(
	stringToTest := UTF8#' ሰማይ አይታረስ ንጉሥ አይከሰስ። ብላ ካለኝ እንደአባቴ በቆመጠኝ።',
	expectedString := UTF8#'አይታረስ ንጉሥ አይከሰስ። ብላ በቆመጠኝ።'
);
THIS^.testisEqualTo(
	stringToTest := UTF8#' ᚻᛖ ᚳᚹᚫᚦ ᚦᚫᛏ ᚻᛖ ᛒᚢᛞᛖ ᚩᚾ ᚦᚫᛗ ᛚᚪᚾᛞᛖ ᚾᚩᚱᚦᚹᛖᚪᚱᛞᚢᛗ ᚹᛁᚦ ᚦᚪ ᚹᛖᛥᚫ',
	expectedString := UTF8#' ᚻᛖ ᚳᚹᚫᚦ ᚦᚫᛏ ᚻᛖ ᛒᚢᛞᛖ ᚩᚾ ᚦᚫᛗ ᛚᚪᚾᛞᛖ ᚾᚩᚱᚦᚹᛖᚪᚱᛞᚢᛗ ᚹᛁᚦ ᚦᚪ ᚹᛖᛥᚫ'
);
THIS^.testisEqualTo(
	stringToTest := UTF8#'⡍⠔⠙⠖ ⡊ ⠙⠕⠝⠰⠞ ⠍⠑⠁⠝ ⠞⠕ ⠎⠁⠹ ⠹⠁⠞ ⡊ ⠅⠝⠪⠂ ⠕⠋ ⠍⠹
  ⠪⠝ ⠅⠝⠪⠇⠫⠛⠑⠂ ⠱⠁⠞ ⠹⠻⠑ ⠊⠎ ⠏⠜⠞⠊⠊⠥⠇⠜⠇⠹ ⠙⠑⠁⠙ ⠁⠃⠳⠞',
	expectedString := UTF8#'⡊ ⠙⠕⠝⠰⠞ ⠍⠑⠁⠝ ⠞⠕ ⠎⠁⠹ ⠹⠁⠞ ⡊ ⠅⠝⠪⠂ ⠕⠋'
);
THIS^.testisEqualTo(
	stringToTest := UTF8#'╔══╦══╗  ┌──┬──┐  ╭──┬──╮  ╭──┬──╮  ┏━━┳━━┓  ┎┒┏┑   ╷  ╻ ┏┯┓ ┌┰┐    ▊ ╱╲╱╲╳╳╳',
	expectedString := UTF8#'╔══╦══╗  ┌──┬──┐  ╭──┬──╮  ╭──┬──╮  ┏━━┳━━┓  ┎┒┏┑   ╷  ╻ ┏┯┓ ┌┰┐    ▊ ╱╲╱╲╳╳╳'
);

THIS^.testisEqualToIgnoreCase(
	stringToTest := 'UPPERCASE',
	expectedString := 'UPPERCASE'
);
THIS^.testisEqualToIgnoreCase(
	stringToTest := 'lowercase',
	expectedString := 'lowercase'
);
THIS^.testisEqualToIgnoreCase(
	stringToTest := 'UPPERCASE',
	expectedString := 'lowercase'
);
THIS^.testisEqualToIgnoreCase(
	stringToTest := 'lowercase',
	expectedString := 'UPPERCASE'
);
THIS^.testisEqualToIgnoreCase(
	stringToTest := UTF8#'UPPERCASE⌷←⍳→⍴∆∇⊃‾⍎⍕⌈',
	expectedString := UTF8#'uppercase⌷←⍳→⍴∆∇⊃‾⍎⍕⌈'
);
THIS^.testisEqualToIgnoreCase(
	stringToTest := UTF8#'UPPERCASE((V⍳V)=⍳⍴V)/V←,V',
	expectedString := UTF8#'uppercase((V⍳V)=⍳⍴V)/V←'
);

TcUnit.TEST_FINISHED();
END_METHOD

(*
short summary
==================
This test method tests ``assert.string.unicode.IsNotEmpty``
method of CNM_AssertionInterfaces library with various inputs

.. <legal notes>

legal notes
=================
| SPDX-FileCopyrightText: © 2022 ekvip automation GmbH <info@ekvip.de>
| SPDX-License-Identifier: Apache-2.0
| For details check: Apache-2.0_

.. _Apache-2.0: https://www.apache.org/licenses/LICENSE-2.0

.. </legal notes>

*)


METHOD runIsNotEmpty : BOOL
VAR_INPUT
END_VAR
RETURN (NOT TcUnit.TEST_ORDERED(THIS^.getTestNameFor('IsNotEmpty')));

THIS^.testIsNotEmpty(
	stringToTest := ''
);
THIS^.testIsNotEmpty(
	stringToTest := 'not empty'
);
THIS^.testIsNotEmpty(
	stringToTest := '{|}~'
);
THIS^.testIsNotEmpty(
	stringToTest := '3649213469328'
);
THIS^.testIsNotEmpty(
	stringToTest := '1one!'
);
THIS^.testIsNotEmpty(
	stringToTest := '$40$n$t$$$"$''
);
THIS^.testIsNotEmpty(
	stringToTest := '$n$t'
);
THIS^.testIsNotEmpty(
	stringToTest := 'frontmiddleback'
);
THIS^.testIsNotEmpty(
	stringToTest := 'backfrontmiddle'
);
THIS^.testIsNotEmpty(
	stringToTest := 'J;%_iTxQSk?6GfWewt}yMKh1)VXqPA@P1YQ:{EAg:8VJ,/FM;j)xJ[[AvYp/}}SzEgtfYS,1K0.5VtA+VJrB(p#55h2z##mw#F)Y@P6Jz9G@6vb=x#E!cYk(Svr@S*KiPJr1VZ6AjrNback4G=vBJd.E:=,k3!wmuGDe#ZKMD#Vx%?M_0&L0#vT]J,+)ZvU{w%8X0=:XzthmT0VG0QrwpXXCWpFxu6[b!c.BunYYfLQi.,?ut?-{jrC1phTHL)y'
);
THIS^.testIsNotEmpty(
	stringToTest := UTF8#'∮ E⋅da = Q,  n → ∞, ∑ f(i) = ∏ g(i), ∀x∈ℝ: ⌈x⌉ = −⌊−x⌋, α ∧ ¬β = ¬(¬α ∨ β)',
);
THIS^.testIsNotEmpty(
	stringToTest := UTF8#'ℕ ⊆ ℕ₀ ⊂ ℤ ⊂ ℚ ⊂ ℝ ⊂ ℂ, ⊥ < a ≠ b ≡ c ≤ d ≪ ⊤ ⇒ (A ⇔ B), 2H₂ + O₂ ⇌ 2H₂O, R = 4.7 kΩ, ⌀ 200 mm',
);
THIS^.testIsNotEmpty(
	stringToTest := UTF8#'ði ıntəˈnæʃənəl fəˈnɛtık əsoʊsiˈeıʃn Y [ˈʏpsilɔn], Yen [jɛn], Yoga [ˈjoːgɑ]',
);
THIS^.testIsNotEmpty(
	stringToTest := UTF8#'‚‘„“‘’“We’ve been here”´` †, ‡, ‰, •, 3–4, —, −5/+5, ™, …, 1lI|, 0OD, 8B, €',
);
THIS^.testIsNotEmpty(
	stringToTest := UTF8#'Σὲ γνωρίζω ἀπὸ τὴν κόψη τοῦ σπαθιοῦ τὴν τρομερή,',
);
THIS^.testIsNotEmpty(
	stringToTest := UTF8#'გთხოვთ ახლავე გაიაროთ რეგისტრაცია Unicode-ის მეათე საერთაშორისო კონფერენციაზე დასასწრებად',
);
THIS^.testIsNotEmpty(
	stringToTest := UTF8#'Зарегистрируйтесь сейчас на Десятую Международную Конференцию по Unicode, которая состоится 10-12 марта 1997 года в',
);
THIS^.testIsNotEmpty(
	stringToTest := UTF8#'๏ แผ่นดินฮั่นเสื่อมโทรมแสนสังเวช  พระปกเกศกองบู๊กู้ขึ้นใหม่'
);
THIS^.testIsNotEmpty(
	stringToTest := UTF8#' ሰማይ አይታረስ ንጉሥ አይከሰስ። ብላ ካለኝ እንደአባቴ በቆመጠኝ።',
);
THIS^.testIsNotEmpty(
	stringToTest := UTF8#' ᚻᛖ ᚳᚹᚫᚦ ᚦᚫᛏ ᚻᛖ ᛒᚢᛞᛖ ᚩᚾ ᚦᚫᛗ ᛚᚪᚾᛞᛖ ᚾᚩᚱᚦᚹᛖᚪᚱᛞᚢᛗ ᚹᛁᚦ ᚦᚪ ᚹᛖᛥᚫ',
);
THIS^.testIsNotEmpty(
	stringToTest := UTF8#'⡍⠔⠙⠖ ⡊ ⠙⠕⠝⠰⠞ ⠍⠑⠁⠝ ⠞⠕ ⠎⠁⠹ ⠹⠁⠞ ⡊ ⠅⠝⠪⠂ ⠕⠋ ⠍⠹
  ⠪⠝ ⠅⠝⠪⠇⠫⠛⠑⠂ ⠱⠁⠞ ⠹⠻⠑ ⠊⠎ ⠏⠜⠞⠊⠊⠥⠇⠜⠇⠹ ⠙⠑⠁⠙ ⠁⠃⠳⠞',
);
THIS^.testIsNotEmpty(
	stringToTest := UTF8#'╔══╦══╗  ┌──┬──┐  ╭──┬──╮  ╭──┬──╮  ┏━━┳━━┓  ┎┒┏┑   ╷  ╻ ┏┯┓ ┌┰┐    ▊ ╱╲╱╲╳╳╳',
);

TcUnit.TEST_FINISHED();
END_METHOD

(*
short summary
==================
This test method tests ``assert.string.unicode.isNotEqualTo``
method of CNM_AssertionInterfaces library with various inputs

.. <legal notes>

legal notes
=================
| SPDX-FileCopyrightText: © 2022 ekvip automation GmbH <info@ekvip.de>
| SPDX-License-Identifier: Apache-2.0
| For details check: Apache-2.0_

.. _Apache-2.0: https://www.apache.org/licenses/LICENSE-2.0

.. </legal notes>

*)


METHOD runIsNotEqualTo : BOOL
VAR_INPUT
END_VAR
RETURN (NOT TcUnit.TEST_ORDERED(THIS^.getTestNameFor('isNotEqualTo')));

THIS^.testisNotEqualTo(
	stringToTest := '',
	expectedString := ''
);
THIS^.testisNotEqualTo(
	stringToTest := 'not empty',
	expectedString := ''
);
THIS^.testisNotEqualTo(
	stringToTest := '',
	expectedString := 'not empty'
);
THIS^.testisNotEqualTo(
	stringToTest := 'not empty',
	expectedString := 'not'
);
THIS^.testisNotEqualTo(
	stringToTest := 'not empty',
	expectedString := 'not empty'
);
THIS^.testisNotEqualTo(
	stringToTest := '{|}~',
	expectedString := '3649213469328'
);
THIS^.testisNotEqualTo(
	stringToTest := '1one!',
	expectedString := '1one'
);
THIS^.testisNotEqualTo(
	stringToTest := '1one!',
	expectedString := '1one!'
);

THIS^.testisNotEqualTo(
	stringToTest := '$40$n$t$$$"$'',
	expectedString := '$n$t'
);
THIS^.testisNotEqualTo(
	stringToTest := '$40$n$t$$$"$'',
	expectedString := '$40$n$t$$$"$''
);
THIS^.testisNotEqualTo(
	stringToTest := 'frontmiddleback',
	expectedString := 'back'
);
THIS^.testisNotEqualTo(
	stringToTest := 'frontmiddleback',
	expectedString := 'frontmiddlebackfront'
);
THIS^.testisNotEqualTo(
	stringToTest := 'backfrontmiddle',
	expectedString := 'backmiddle'
);
THIS^.testisNotEqualTo(
	stringToTest := 'J;%_iTxQSk?6GfWewt}yMKh1)VXqPA@P1YQ:{EAg:8VJ,/FM;j)xJ[[AvYp/}}SzEgtfYS,1K0.5VtA+VJrB(p#55h2z##mw#F)Y@P6Jz9G@6vb=x#E!cYk(Svr@S*KiPJr1VZ6AjrNback4G=vBJd.E:=,k3!wmuGDe#ZKMD#Vx%?M_0&L0#vT]J,+)ZvU{w%8X0=:XzthmT0VG0QrwpXXCWpFxu6[b!c.BunYYfLQi.,?ut?-{jrC1phTHL)y',
	expectedString := 'J;%_iTxQSk?6GfWewt}yMKh1)VXqPA@P1YQ:{EAg:8VJ,/FM;j)xJ[[AvYp/}}SzEgtfYS,1K0.5VtA+VJrB(p#55h2z##mw#F)Y@P6Jz9G@6vb=x#E!cYk(Svr@S*KiPJr1VZ6AjrNback4G=vBJd.E:=,k3!wmuGDe#ZKMD#Vx%?M_0&L0#vT]J,+)ZvU{w%8X0=:XzthmT0VG0QrwpXXCWpFxu6[b!c.BunYYfLQi.,?ut?-{jrC1phTHL)y'
);
THIS^.testisNotEqualTo(
	stringToTest := 'J;%_iTxQSk?6GfWewt}yMKh1)VXqPA@P1YQ:{EAg:8VJ,/FM;j)xJ[[AvYp/}}SzEgtfYS,1K0.5VtA+VJrB(p#55h2z##mw#F)Y@P6Jz9G@6vb=x#E!cYk(Svr@S*KiPJr1VZ6AjrNback4G=vBJd.E:=,k3!wmuGDe#ZKMD#Vx%?M_0&L0#vT]J,+)ZvU{w%8X0=:XzthmT0VG0QrwpXXCWpFxu6[b!c.BunYYfLQi.,?ut?-{jrC1phTHL)y',
	expectedString := 'J;%_iTxQSk?6GfWewt}yMKh1)VXqPA@P1YQ:{EAg:8VJ,/FM;j)xJ[[AvYp/}}SzEgtfYS,1K0.5VtA+VJrB(p#55h2z##mw#F)Y@P6Jz9G@6vb=x#E!cYk(Svr@S*KiPJr1VZ6AjrNback4G=vBJd.E:=,k3!wmuGDe#ZKMD#Vx%?M_0&L0#vT]J,+)ZvU{w%8X0=:XzthmT0VG0QrwpXXCWpFxu6[b!c.BunYYfLQi.,?ut?-{jrC1phTHL)x'
);
THIS^.testisNotEqualTo(
	stringToTest := UTF8#'∮ E⋅da = Q,  n → ∞, ∑ f(i) = ∏ g(i), ∀x∈ℝ: ⌈x⌉ = −⌊−x⌋, α ∧ ¬β = ¬(¬α ∨ β)',
	expectedString := UTF8#'∮ E⋅da = Q,  n → ∞, ∑ f(i) = ∏ g(i), ∀x∈ℝ: ⌈x⌉ = −⌊−x⌋, α ∧ ¬β = ¬(¬α ∨ β)'
);
THIS^.testisNotEqualTo(
	stringToTest := UTF8#'ℕ ⊆ ℕ₀ ⊂ ℤ ⊂ ℚ ⊂ ℝ ⊂ ℂ, ⊥ < a ≠ b ≡ c ≤ d ≪ ⊤ ⇒ (A ⇔ B), 2H₂ + O₂ ⇌ 2H₂O, R = 4.7 kΩ, ⌀ 200 mm',
	expectedString := UTF8#'ℕ ⊆ ℕ₀ ⊂ ℤ ⊂ ℚ ⊂ ℝ ⊂ ℂ'
);
THIS^.testisNotEqualTo(
	stringToTest := UTF8#'ℕ ⊆ ℕ₀ ⊂ ℤ ⊂ ℚ ⊂ ℝ ⊂ ℂ, ⊥ < a ≠ b ≡ c ≤ d ≪ ⊤ ⇒ (A ⇔ B), 2H₂ + O₂ ⇌ 2H₂O, R = 4.7 kΩ, ⌀ 200 mm',
	expectedString := UTF8#'ℕ ⊆ ℕ₀ ⊂ ℤ ⊂ ℚ ⊂ ℝ ⊂ ℂ, ⊥ < a ≠ b ≡ c ≤ d ≪ ⊤ ⇒ (A ⇔ B), 2H₂ + O₂ ⇌ 2H₂O, R = 4.7 kΩ, ⌀ 200 mm'
);
THIS^.testisNotEqualTo(
	stringToTest := UTF8#'ði ıntəˈnæʃənəl fəˈnɛtık əsoʊsiˈeıʃn Y [ˈʏpsilɔn], Yen [jɛn], Yoga [ˈjoːgɑ]',
	expectedString := UTF8#'ˈnæʃənəl fəˈnɛtık '
);
THIS^.testisNotEqualTo(
	stringToTest := UTF8#'‚‘„“‘’“We’ve been here”´` †, ‡, ‰, •, 3–4, —, −5/+5, ™, …, 1lI|, 0OD, 8B, €',
	expectedString := UTF8#'‚‘„“‘’“We’ve been here”´` †, ‡, ‰, •, 3–4, —, −5/+5, ™, …, 1lI|, 0OD, 8B, €'
);
THIS^.testisNotEqualTo(
	stringToTest := UTF8#'Σὲ γνωρίζω ἀπὸ τὴν κόψη τοῦ σπαθιοῦ τὴν τρομερή,',
	expectedString := UTF8#'τὴν κόψη τοῦ σπαθ'
);
THIS^.testisNotEqualTo(
	stringToTest := UTF8#'გთხოვთ ახლავე გაიაროთ რეგისტრაცია Unicode-ის მეათე საერთაშორისო კონფერენციაზე დასასწრებად',
	expectedString := UTF8#'გთხოვთ ახლავე გაიაროთ რეგისტრაცია Unicode-ის მეათე საერთაშორისო კონფერენციაზე დასასწრებად'
);
THIS^.testisNotEqualTo(
	stringToTest := UTF8#'Зарегистрируйтесь сейчас на Десятую Международную Конференцию по Unicode, которая состоится 10-12 марта 1997 года в',
	expectedString := UTF8#'Международную Конференцию по Unicode, которая'
);
THIS^.testisNotEqualTo(
	stringToTest := UTF8#'๏ แผ่นดินฮั่นเสื่อมโทรมแสนสังเวช  พระปกเกศกองบู๊กู้ขึ้นใหม่',
	expectedString := UTF8#'๏ แผ่นดินฮั่นเสื่อมโทรมแสนสังเวช  พระปกเกศกองบู๊กู้ขึ้นใหม่'
);
THIS^.testisNotEqualTo(
	stringToTest := UTF8#' ሰማይ አይታረስ ንጉሥ አይከሰስ። ብላ ካለኝ እንደአባቴ በቆመጠኝ።',
	expectedString := UTF8#'አይታረስ ንጉሥ አይከሰስ። ብላ በቆመጠኝ።'
);
THIS^.testisNotEqualTo(
	stringToTest := UTF8#' ᚻᛖ ᚳᚹᚫᚦ ᚦᚫᛏ ᚻᛖ ᛒᚢᛞᛖ ᚩᚾ ᚦᚫᛗ ᛚᚪᚾᛞᛖ ᚾᚩᚱᚦᚹᛖᚪᚱᛞᚢᛗ ᚹᛁᚦ ᚦᚪ ᚹᛖᛥᚫ',
	expectedString := UTF8#' ᚻᛖ ᚳᚹᚫᚦ ᚦᚫᛏ ᚻᛖ ᛒᚢᛞᛖ ᚩᚾ ᚦᚫᛗ ᛚᚪᚾᛞᛖ ᚾᚩᚱᚦᚹᛖᚪᚱᛞᚢᛗ ᚹᛁᚦ ᚦᚪ ᚹᛖᛥᚫ'
);
THIS^.testisNotEqualTo(
	stringToTest := UTF8#'⡍⠔⠙⠖ ⡊ ⠙⠕⠝⠰⠞ ⠍⠑⠁⠝ ⠞⠕ ⠎⠁⠹ ⠹⠁⠞ ⡊ ⠅⠝⠪⠂ ⠕⠋ ⠍⠹
  ⠪⠝ ⠅⠝⠪⠇⠫⠛⠑⠂ ⠱⠁⠞ ⠹⠻⠑ ⠊⠎ ⠏⠜⠞⠊⠊⠥⠇⠜⠇⠹ ⠙⠑⠁⠙ ⠁⠃⠳⠞',
	expectedString := UTF8#'⡊ ⠙⠕⠝⠰⠞ ⠍⠑⠁⠝ ⠞⠕ ⠎⠁⠹ ⠹⠁⠞ ⡊ ⠅⠝⠪⠂ ⠕⠋'
);
THIS^.testisNotEqualTo(
	stringToTest := UTF8#'╔══╦══╗  ┌──┬──┐  ╭──┬──╮  ╭──┬──╮  ┏━━┳━━┓  ┎┒┏┑   ╷  ╻ ┏┯┓ ┌┰┐    ▊ ╱╲╱╲╳╳╳',
	expectedString := UTF8#'╔══╦══╗  ┌──┬──┐  ╭──┬──╮  ╭──┬──╮  ┏━━┳━━┓  ┎┒┏┑   ╷  ╻ ┏┯┓ ┌┰┐    ▊ ╱╲╱╲╳╳╳'
);

THIS^.testisNotEqualToIgnoreCase(
	stringToTest := 'UPPERCASE',
	expectedString := 'UPPERCASE'
);
THIS^.testisNotEqualToIgnoreCase(
	stringToTest := 'lowercase',
	expectedString := 'lowercase'
);
THIS^.testisNotEqualToIgnoreCase(
	stringToTest := 'UPPERCASE',
	expectedString := 'lowercase'
);
THIS^.testisNotEqualToIgnoreCase(
	stringToTest := 'lowercase',
	expectedString := 'UPPERCASE'
);
THIS^.testisNotEqualToIgnoreCase(
	stringToTest := UTF8#'UPPERCASE⌷←⍳→⍴∆∇⊃‾⍎⍕⌈',
	expectedString := UTF8#'uppercase⌷←⍳→⍴∆∇⊃‾⍎⍕⌈'
);
THIS^.testisNotEqualToIgnoreCase(
	stringToTest := UTF8#'UPPERCASE((V⍳V)=⍳⍴V)/V←,V',
	expectedString := UTF8#'uppercase((V⍳V)=⍳⍴V)/V←'
);

TcUnit.TEST_FINISHED();
END_METHOD

(*
short summary
==================
This test method tests ``assert.string.unicode.lengthIsBetween``
method of CNM_AssertionInterfaces library with various inputs

.. <legal notes>

legal notes
=================
| SPDX-FileCopyrightText: © 2022 ekvip automation GmbH <info@ekvip.de>
| SPDX-License-Identifier: Apache-2.0
| For details check: Apache-2.0_

.. _Apache-2.0: https://www.apache.org/licenses/LICENSE-2.0

.. </legal notes>

*)


METHOD runLengthIsBetween : BOOL
VAR
	(* for the test it's the parameter ``stringToCheck`` *)
	{attribute 'TcEncoding' := 'UTF-8'}
	stringToTest :Tc2_System.T_MaxString;
	(* length of current string to check in bytes *)
	stringToTestByteCount		:UDINT;
	(* length of current string to check in characters *)
	stringToTestCodePointCount	:UDINT;
	(* length of ´´stringToCheck´´ *)
	normalizedLength :UDINT;
	(* holds the normalized ´´stringToCheck´´ *)
	{attribute 'TcEncoding' := 'UTF-8'}
	normalizedStringToTest :Tc2_System.T_MaxString;
	(* width of ´´stringToCheck´´ *)
	stringToTestWidth :DINT;
	(* visible characters of ´´stringToCheck´´ *)
	stringToTestVisibleCharacters :UDINT := 0;
END_VAR
RETURN (NOT TcUnit.TEST_ORDERED(THIS^.getTestNameFor('lengthIsBetween')));

THIS^.testLengthIsBetween(
	stringToTest := '',
	maxLength := 0,
	minLength := 0,
	stringLengthUnit := CNM_AssertionInterfaces.UnicodeStringLengthUnit.BYTES
);
THIS^.testLengthIsBetween(
	stringToTest := '',
	maxLength := 0,
	minLength := 1,
	stringLengthUnit := CNM_AssertionInterfaces.UnicodeStringLengthUnit.BYTES
);
THIS^.testLengthIsBetween(
	stringToTest := '',
	maxLength := 0,
	minLength := 0,
	stringLengthUnit := CNM_AssertionInterfaces.UnicodeStringLengthUnit.CHARACTERS
);
THIS^.testLengthIsBetween(
	stringToTest := '',
	maxLength := 0,
	minLength := 1,
	stringLengthUnit := CNM_AssertionInterfaces.UnicodeStringLengthUnit.CHARACTERS
);
THIS^.testLengthIsBetween(
	stringToTest := 'not empty',
	maxLength := 9,
	minLength := 0,
	stringLengthUnit := CNM_AssertionInterfaces.UnicodeStringLengthUnit.CHARACTERS
);
THIS^.testLengthIsBetween(
	stringToTest := 'not empty',
	maxLength := 13,
	minLength := 10,
	stringLengthUnit := CNM_AssertionInterfaces.UnicodeStringLengthUnit.CHARACTERS
);
THIS^.testLengthIsBetween(
	stringToTest := 'not empty',
	maxLength := 9,
	minLength := 9,
	stringLengthUnit := CNM_AssertionInterfaces.UnicodeStringLengthUnit.BYTES
);
THIS^.testLengthIsBetween(
	stringToTest := 'not empty',
	maxLength := 13,
	minLength := 10,
	stringLengthUnit := CNM_AssertionInterfaces.UnicodeStringLengthUnit.BYTES
);
THIS^.testLengthIsBetween(
	stringToTest := '1one!',
	maxLength := 5,
	minLength := 4,
	stringLengthUnit := CNM_AssertionInterfaces.UnicodeStringLengthUnit.VISIBLE_CHARACTERS
);
THIS^.testLengthIsBetween(
	stringToTest := '1one!',
	maxLength := 5,
	minLength := 4,
	stringLengthUnit := CNM_AssertionInterfaces.UnicodeStringLengthUnit.WIDTH
);
THIS^.testLengthIsBetween(
	stringToTest := 'J;%_iTxQSk?6GfWewt}yMKh1)VXqPA@P1YQ:{EAg:8VJ,/FM;j)xJ[[AvYp/}}SzEgtfYS,1K0.5VtA+VJrB(p#55h2z##mw#F)Y@P6Jz9G@6vb=x#E!cYk(Svr@S*KiPJr1VZ6AjrNback4G=vBJd.E:=,k3!wmuGDe#ZKMD#Vx%?M_0&L0#vT]J,+)ZvU{w%8X0=:XzthmT0VG0QrwpXXCWpFxu6[b!c.BunYYfLQi.,?ut?-{jrC1phTHL)y',
	maxLength := 255,
	minLength := 255,
	stringLengthUnit := CNM_AssertionInterfaces.UnicodeStringLengthUnit.CHARACTERS
);
THIS^.testLengthIsBetween(
	stringToTest := 'J;%_iTxQSk?6GfWewt}yMKh1)VXqPA@P1YQ:{EAg:8VJ,/FM;j)xJ[[AvYp/}}SzEgtfYS,1K0.5VtA+VJrB(p#55h2z##mw#F)Y@P6Jz9G@6vb=x#E!cYk(Svr@S*KiPJr1VZ6AjrNback4G=vBJd.E:=,k3!wmuGDe#ZKMD#Vx%?M_0&L0#vT]J,+)ZvU{w%8X0=:XzthmT0VG0QrwpXXCWpFxu6[b!c.BunYYfLQi.,?ut?-{jrC1phTHL)y',
	maxLength := 255,
	minLength := 255,
	stringLengthUnit := CNM_AssertionInterfaces.UnicodeStringLengthUnit.BYTES
);
THIS^.testLengthIsBetween(
	stringToTest := 'J;%_iTxQSk?6GfWewt}yMKh1)VXqPA@P1YQ:{EAg:8VJ,/FM;j)xJ[[AvYp/}}SzEgtfYS,1K0.5VtA+VJrB(p#55h2z##mw#F)Y@P6Jz9G@6vb=x#E!cYk(Svr@S*KiPJr1VZ6AjrNback4G=vBJd.E:=,k3!wmuGDe#ZKMD#Vx%?M_0&L0#vT]J,+)ZvU{w%8X0=:XzthmT0VG0QrwpXXCWpFxu6[b!c.BunYYfLQi.,?ut?-{jrC1phTHL)y',
	maxLength := 254,
	minLength := 0,
	stringLengthUnit := CNM_AssertionInterfaces.UnicodeStringLengthUnit.CHARACTERS
);
THIS^.testLengthIsBetween(
	stringToTest := 'J;%_iTxQSk?6GfWewt}yMKh1)VXqPA@P1YQ:{EAg:8VJ,/FM;j)xJ[[AvYp/}}SzEgtfYS,1K0.5VtA+VJrB(p#55h2z##mw#F)Y@P6Jz9G@6vb=x#E!cYk(Svr@S*KiPJr1VZ6AjrNback4G=vBJd.E:=,k3!wmuGDe#ZKMD#Vx%?M_0&L0#vT]J,+)ZvU{w%8X0=:XzthmT0VG0QrwpXXCWpFxu6[b!c.BunYYfLQi.,?ut?-{jrC1phTHL)y',
	maxLength := 254,
	minLength := 254,
	stringLengthUnit := CNM_AssertionInterfaces.UnicodeStringLengthUnit.BYTES
);

stringToTest := UTF8#'∮ E⋅da = Q,  n → ∞, ∑ f(i) = ∏ g(i), ∀x∈ℝ: ⌈x⌉ = −⌊−x⌋, α ∧ ¬β = ¬(¬α ∨ β)';
CNM_UnicodeUtilities.GetUtf8StringLength(ADR(stringToTest), byteCount => stringToTestByteCount, characterCount => stringToTestCodePointCount,);
CNM_UnicodeUtilities.GetUtf8StringWidth(ADR(stringToTest), visibleCharacters => stringToTestVisibleCharacters, width => stringToTestWidth);
THIS^.testLengthIsBetween(
	stringToTest := stringToTest,
	maxLength := stringToTestByteCount,
	minLength := stringToTestByteCount,
	stringLengthUnit := CNM_AssertionInterfaces.UnicodeStringLengthUnit.BYTES,
	stringToTestPrintable := 'S E*da = Q,  n > inf ...'
);
THIS^.testLengthIsBetween(
	stringToTest := stringToTest,
	maxLength := stringToTestCodePointCount,
	minLength := stringToTestCodePointCount,
	stringLengthUnit := CNM_AssertionInterfaces.UnicodeStringLengthUnit.CHARACTERS,
	stringToTestPrintable := 'S E*da = Q,  n > inf ...'
);
THIS^.testLengthIsBetween(
	stringToTest := stringToTest,
	maxLength := stringToTestByteCount - 1,
	minLength := 0,
	stringLengthUnit := CNM_AssertionInterfaces.UnicodeStringLengthUnit.CHARACTERS,
	stringToTestPrintable := 'S E*da = Q,  n > inf ...'
);
THIS^.testLengthIsBetween(
	stringToTest := stringToTest,
	maxLength := TO_UDINT(stringToTestWidth),
	minLength := TO_UDINT(stringToTestWidth),
	stringLengthUnit := CNM_AssertionInterfaces.UnicodeStringLengthUnit.WIDTH,
	stringToTestPrintable := 'S E*da = Q,  n > inf ...'
);
THIS^.testLengthIsBetween(
	stringToTest := stringToTest,
	maxLength := stringToTestVisibleCharacters,
	minLength := stringToTestVisibleCharacters,
	stringLengthUnit := CNM_AssertionInterfaces.UnicodeStringLengthUnit.VISIBLE_CHARACTERS,
	stringToTestPrintable := 'S E*da = Q,  n > inf ...'
);

stringToTest := UTF8#'Зарегистрируйтесь сейчас на Десятую Международную Конференцию по Unicode, которая состоится 10-12 марта 1997 года в';
CNM_UnicodeUtilities.GetUtf8StringLength(ADR(stringToTest), byteCount => stringToTestByteCount, characterCount => stringToTestCodePointCount,);
CNM_UnicodeUtilities.GetUtf8StringWidth(ADR(stringToTest), visibleCharacters => stringToTestVisibleCharacters, width => stringToTestWidth);
THIS^.testLengthIsBetween(
	stringToTest := stringToTest,
	maxLength := stringToTestByteCount,
	minLength := stringToTestByteCount,
	stringLengthUnit := CNM_AssertionInterfaces.UnicodeStringLengthUnit.BYTES,
	stringToTestPrintable := 'Zaregistriruytes$' seychas ...'
);
THIS^.testLengthIsBetween(
	stringToTest := stringToTest,
	maxLength := stringToTestCodePointCount,
	minLength := stringToTestCodePointCount,
	stringLengthUnit := CNM_AssertionInterfaces.UnicodeStringLengthUnit.CHARACTERS,
	stringToTestPrintable := 'Zaregistriruytes$' seychas ...'
);
THIS^.testLengthIsBetween(
	stringToTest := stringToTest,
	maxLength := stringToTestCodePointCount + 1,
	minLength := stringToTestCodePointCount - 1,
	stringLengthUnit := CNM_AssertionInterfaces.UnicodeStringLengthUnit.CHARACTERS,
	stringToTestPrintable := 'Zaregistriruytes$' seychas ...'
);
THIS^.testLengthIsBetween(
	stringToTest := stringToTest,
	maxLength := TO_UDINT(stringToTestWidth),
	minLength := TO_UDINT(stringToTestWidth),
	stringLengthUnit := CNM_AssertionInterfaces.UnicodeStringLengthUnit.WIDTH,
	stringToTestPrintable := 'Zaregistriruytes$' seychas ...'
); 
THIS^.testLengthIsBetween(
	stringToTest := stringToTest,
	maxLength := stringToTestVisibleCharacters,
	minLength := stringToTestVisibleCharacters,
	stringLengthUnit := CNM_AssertionInterfaces.UnicodeStringLengthUnit.VISIBLE_CHARACTERS,
	stringToTestPrintable := 'Zaregistriruytes$' seychas ...'
);
CNM_UnicodeUtilities.NormalizeUtf8String(
	utf8StringBuffer := ADR(stringToTest),
	normalForm := CNM_UnicodeUtilities.NormalizationForm.NFD,
	normalizedStringBuffer := ADR(normalizedStringToTest),
	bufferSize := Tc2_System.MAX_STRING_LENGTH + 1,
	normalizedStringLength => normalizedLength
);
CNM_UnicodeUtilities.GetUtf8StringLength(
	stringAddress := ADR(normalizedStringToTest),
	characterCount => stringToTestCodePointCount
);
THIS^.testLengthIsBetween(
	stringToTest := stringToTest,
	maxLength := stringToTestCodePointCount,
	minLength := stringToTestCodePointCount,
	stringLengthUnit := CNM_AssertionInterfaces.UnicodeStringLengthUnit.CHARACTERS_NFD,
	stringToTestPrintable := 'Zaregistriruytes$' seychas ...'
);
CNM_UnicodeUtilities.NormalizeUtf8String(
	utf8StringBuffer := ADR(stringToTest),
	normalForm := CNM_UnicodeUtilities.NormalizationForm.NFC,
	normalizedStringBuffer := ADR(normalizedStringToTest),
	bufferSize := Tc2_System.MAX_STRING_LENGTH + 1,
	normalizedStringLength => normalizedLength
);
CNM_UnicodeUtilities.GetUtf8StringLength(
	stringAddress := ADR(normalizedStringToTest),
	characterCount => stringToTestCodePointCount
);
THIS^.testLengthIsBetween(
	stringToTest := stringToTest,
	maxLength := stringToTestCodePointCount,
	minLength := stringToTestCodePointCount,
	stringLengthUnit := CNM_AssertionInterfaces.UnicodeStringLengthUnit.CHARACTERS_NFC,
	stringToTestPrintable := 'Zaregistriruytes$' seychas ...'
);
THIS^.testLengthIsBetween(
	stringToTest := stringToTest,
	maxLength := stringToTestCodePointCount,
	minLength := stringToTestCodePointCount,
	stringLengthUnit := CNM_AssertionInterfaces.UnicodeStringLengthUnit.CHARACTERS_NFD,
	stringToTestPrintable := 'Zaregistriruytes$' seychas ...'
);

stringToTest := UTF8#'Ä๏ แผ่นดินฮั่นเสื่อมโทรมแสนสังเวช  พระปกเกศกองบู๊กู้ขึ้นใหม่  สิบสองกษัตริย์ก่อนหน้าแล ';
CNM_UnicodeUtilities.GetUtf8StringLength(ADR(stringToTest), byteCount => stringToTestByteCount, characterCount => stringToTestCodePointCount,);
CNM_UnicodeUtilities.GetUtf8StringWidth(ADR(stringToTest), visibleCharacters => stringToTestVisibleCharacters, width => stringToTestWidth);
THIS^.testLengthIsBetween(
	stringToTest := stringToTest,
  	maxLength := stringToTestByteCount,
  	minLength := stringToTestByteCount,
	stringLengthUnit := CNM_AssertionInterfaces.UnicodeStringLengthUnit.BYTES,
 	stringToTestPrintable := '* aephndinhanesueomothrmaesnsangewch  ...'
);
THIS^.testLengthIsBetween(
	stringToTest := stringToTest,
 	maxLength := stringToTestCodePointCount,
 	minLength := stringToTestCodePointCount,
	stringLengthUnit := CNM_AssertionInterfaces.UnicodeStringLengthUnit.CHARACTERS,
  	stringToTestPrintable := '* aephndinhanesueomothrmaesnsangewch  ...'
);
THIS^.testLengthIsBetween(
	stringToTest := stringToTest,
 	maxLength := TO_UDINT(stringToTestWidth),
  	minLength := TO_UDINT(stringToTestWidth),
	stringLengthUnit := CNM_AssertionInterfaces.UnicodeStringLengthUnit.WIDTH,
 	stringToTestPrintable := '* aephndinhanesueomothrmaesnsangewch  ...'
);
THIS^.testLengthIsBetween(
	stringToTest := stringToTest,
  	maxLength := stringToTestVisibleCharacters,
  	minLength := stringToTestVisibleCharacters,
	stringLengthUnit := CNM_AssertionInterfaces.UnicodeStringLengthUnit.VISIBLE_CHARACTERS,
  	stringToTestPrintable := '* aephndinhanesueomothrmaesnsangewch  ...'
);
CNM_UnicodeUtilities.NormalizeUtf8String(
	utf8StringBuffer := ADR(stringToTest),
	normalForm := CNM_UnicodeUtilities.NormalizationForm.NFD,
	normalizedStringBuffer := ADR(normalizedStringToTest),
	bufferSize := Tc2_System.MAX_STRING_LENGTH + 1,
	normalizedStringLength => normalizedLength
);
CNM_UnicodeUtilities.GetUtf8StringLength(
	stringAddress := ADR(normalizedStringToTest),
	characterCount => stringToTestCodePointCount
);
THIS^.testLengthIsBetween(
	stringToTest := stringToTest,
  	maxLength := stringToTestCodePointCount,
  	minLength := stringToTestCodePointCount,
	stringLengthUnit := CNM_AssertionInterfaces.UnicodeStringLengthUnit.CHARACTERS_NFD,
  	stringToTestPrintable := '* aephndinhanesueomothrmaesnsangewch  ...'
);
CNM_UnicodeUtilities.NormalizeUtf8String(
	utf8StringBuffer := ADR(stringToTest),
	normalForm := CNM_UnicodeUtilities.NormalizationForm.NFC,
	normalizedStringBuffer := ADR(normalizedStringToTest),
	bufferSize := Tc2_System.MAX_STRING_LENGTH + 1,
	normalizedStringLength => normalizedLength
);
CNM_UnicodeUtilities.GetUtf8StringLength(
	stringAddress := ADR(normalizedStringToTest),
	characterCount => stringToTestCodePointCount
);
THIS^.testLengthIsBetween(
	stringToTest := stringToTest,
  	maxLength := stringToTestCodePointCount,
  	minLength := stringToTestCodePointCount,
	stringLengthUnit := CNM_AssertionInterfaces.UnicodeStringLengthUnit.CHARACTERS_NFC,
  	stringToTestPrintable := '* aephndinhanesueomothrmaesnsangewch  ...'
);
THIS^.testLengthIsBetween(
	stringToTest := stringToTest,
  	maxLength := stringToTestCodePointCount,
  	minLength := stringToTestCodePointCount,
	stringLengthUnit := CNM_AssertionInterfaces.UnicodeStringLengthUnit.CHARACTERS_NFD,
  	stringToTestPrintable := '* aephndinhanesueomothrmaesnsangewch  ...'
);

stringToTest := UTF8#'🧌🦤🏭💽🧧🪷👨‍💻👩‍👩‍👧‍👦';
CNM_UnicodeUtilities.GetUtf8StringLength(ADR(stringToTest), byteCount => stringToTestByteCount, characterCount => stringToTestCodePointCount,);
CNM_UnicodeUtilities.GetUtf8StringWidth(ADR(stringToTest), visibleCharacters => stringToTestVisibleCharacters, width => stringToTestWidth);
THIS^.testLengthIsBetween(
	stringToTest := stringToTest,
  	maxLength := stringToTestByteCount,
  	minLength := stringToTestByteCount,
	stringLengthUnit := CNM_AssertionInterfaces.UnicodeStringLengthUnit.BYTES,
  	stringToTestPrintable := ':troll::dodo::factory:...'
);
THIS^.testLengthIsBetween(
	stringToTest := stringToTest,
  	maxLength := stringToTestCodePointCount,
  	minLength := stringToTestCodePointCount,
	stringLengthUnit := CNM_AssertionInterfaces.UnicodeStringLengthUnit.CHARACTERS,
  	stringToTestPrintable := ':troll::dodo::factory:...'
);
THIS^.testLengthIsBetween(
	stringToTest := stringToTest,
  	maxLength := stringToTestCodePointCount + 1,
  	minLength := stringToTestCodePointCount - 1,
	stringLengthUnit := CNM_AssertionInterfaces.UnicodeStringLengthUnit.CHARACTERS,
  	stringToTestPrintable := ':troll::dodo::factory:...'
);
THIS^.testLengthIsBetween(
	stringToTest := stringToTest,
  	maxLength := TO_UDINT(stringToTestWidth),
  	minLength := TO_UDINT(stringToTestWidth),
	stringLengthUnit := CNM_AssertionInterfaces.UnicodeStringLengthUnit.WIDTH,
  	stringToTestPrintable := ':troll::dodo::factory:...'
);
THIS^.testLengthIsBetween(
	stringToTest := stringToTest,
  	maxLength := stringToTestVisibleCharacters,
  	minLength := stringToTestVisibleCharacters,
	stringLengthUnit := CNM_AssertionInterfaces.UnicodeStringLengthUnit.VISIBLE_CHARACTERS,
  	stringToTestPrintable := ':troll::dodo::factory:...'
);
CNM_UnicodeUtilities.NormalizeUtf8String(
	utf8StringBuffer := ADR(stringToTest),
	normalForm := CNM_UnicodeUtilities.NormalizationForm.NFD,
	normalizedStringBuffer := ADR(normalizedStringToTest),
	bufferSize := Tc2_System.MAX_STRING_LENGTH + 1,
	normalizedStringLength => normalizedLength
);
CNM_UnicodeUtilities.GetUtf8StringLength(
	stringAddress := ADR(normalizedStringToTest),
	characterCount => stringToTestCodePointCount
);
THIS^.testLengthIsBetween(
	stringToTest := stringToTest,
  	maxLength := stringToTestCodePointCount,
  	minLength := stringToTestCodePointCount,
	stringLengthUnit := CNM_AssertionInterfaces.UnicodeStringLengthUnit.CHARACTERS_NFD,
  	stringToTestPrintable := ':troll::dodo::factory:...'
);
CNM_UnicodeUtilities.NormalizeUtf8String(
	utf8StringBuffer := ADR(stringToTest),
	normalForm := CNM_UnicodeUtilities.NormalizationForm.NFC,
	normalizedStringBuffer := ADR(normalizedStringToTest),
	bufferSize := Tc2_System.MAX_STRING_LENGTH + 1,
	normalizedStringLength => normalizedLength
);
CNM_UnicodeUtilities.GetUtf8StringLength(
	stringAddress := ADR(normalizedStringToTest),
	characterCount => stringToTestCodePointCount
);
THIS^.testLengthIsBetween(
	stringToTest := stringToTest,
  	maxLength := stringToTestCodePointCount,
  	minLength := stringToTestCodePointCount,
	stringLengthUnit := CNM_AssertionInterfaces.UnicodeStringLengthUnit.CHARACTERS_NFC,
  	stringToTestPrintable := ':troll::dodo::factory:...'
);

TcUnit.TEST_FINISHED();
END_METHOD

(*
short summary
==================
This test method tests ``assert.string.unicode.lengthIsExact``
method of CNM_AssertionInterfaces library with various inputs

.. <legal notes>

legal notes
=================
| SPDX-FileCopyrightText: © 2022 ekvip automation GmbH <info@ekvip.de>
| SPDX-License-Identifier: Apache-2.0
| For details check: Apache-2.0_

.. _Apache-2.0: https://www.apache.org/licenses/LICENSE-2.0

.. </legal notes>

*)


